(* IEC 61131-3 sources: AXOpen/src/components.dukane.welders/ctrl/src/Axo_IQ_SeriesWelder (part 2) *)

        METHOD PRIVATE ByteArray_TO_buf4
            VAR_INPUT
                array_buffer : ARRAY[0..253] OF BYTE;
            END_VAR
            VAR_IN_OUT
                buf4 : Axo_IQ_SeriesWelder_data4_200bytes;
            END_VAR
			buf4.Weld2Distance.Enable._0 						    :=   array_buffer[  0].%X0;
			buf4.Weld2Distance.Enable._1 						    :=   array_buffer[  0].%X1;
			buf4.Weld2Distance.Enable._2 						    :=   array_buffer[  0].%X2;
			buf4.Weld2Distance.Enable._3 						    :=   array_buffer[  0].%X3;
			buf4.Weld2Distance.Enable._4 						    :=   array_buffer[  0].%X4;
			buf4.Weld2Distance.Enable._5 						    :=   array_buffer[  0].%X5;
			buf4.Weld2Distance.Enable._6 						    :=   array_buffer[  0].%X6;
			buf4.Weld2Distance.Enable._7 						    :=   array_buffer[  0].%X7;
			buf4.Weld2Distance.Enable._8 						    :=   array_buffer[  1].%X0;
			buf4.Weld2Distance.Enable._9 						    :=   array_buffer[  1].%X1;
			buf4.Weld2Distance.Enable._10 					        :=   array_buffer[  1].%X2;
			buf4.Weld2Distance.Enable._11 					        :=   array_buffer[  1].%X3;
			buf4.Weld2Distance.Enable._12 					        :=   array_buffer[  1].%X4;
			buf4.Weld2Distance.Enable._13 					        :=   array_buffer[  1].%X5;
			buf4.Weld2Distance.Enable._14 					        :=   array_buffer[  1].%X6;
			buf4.Weld2Distance.Enable._15 					        :=   array_buffer[  1].%X7;
			buf4.Weld2Distance.Enable._16 					        :=   array_buffer[  2].%X0;
			buf4.Weld2Distance.Enable._17 					        :=   array_buffer[  2].%X1;
			buf4.Weld2Distance.Enable._18 					        :=   array_buffer[  2].%X2;
			buf4.Weld2Distance.Enable._19 					        :=   array_buffer[  2].%X3;
			buf4.Weld2Distance.Enable._20 					        :=   array_buffer[  2].%X4;
			buf4.Weld2Distance.Enable._21 					        :=   array_buffer[  2].%X5;
			buf4.Weld2Distance.Enable._22 					        :=   array_buffer[  2].%X6;
			buf4.Weld2Distance.Enable._23 					        :=   array_buffer[  2].%X7;
			buf4.Weld2Distance.Enable.LowerBad_1 				    :=   array_buffer[  3].%X0;
			buf4.Weld2Distance.Enable.LowerSuspect_1 			    :=   array_buffer[  3].%X1;
			buf4.Weld2Distance.Enable.UpperSuspect_1			    :=   array_buffer[  3].%X2;
			buf4.Weld2Distance.Enable.UpperBad_1 				    :=   array_buffer[  3].%X3;
			buf4.Weld2Distance.Enable.Display_1 				    :=   array_buffer[  3].%X4;
			buf4.Weld2Distance.Enable._29 					        :=   array_buffer[  3].%X5;
			buf4.Weld2Distance.Enable._30 					        :=   array_buffer[  3].%X6;
			buf4.Weld2Distance.Enable._31 					        :=   array_buffer[  3].%X7;
			buf4.Weld2Distance.LowerBad:=           TO_DINT(SHL(TO_DWORD(array_buffer[  4]), UINT#24) OR
															SHL(TO_DWORD(array_buffer[  5]), UINT#16) OR
															SHL(TO_DWORD(array_buffer[  6]),  UINT#8) OR
																TO_DWORD(array_buffer[  7]));
			buf4.Weld2Distance.LowerSuspect:=       TO_DINT(SHL(TO_DWORD(array_buffer[  8]), UINT#24) OR
															SHL(TO_DWORD(array_buffer[  9]), UINT#16) OR
															SHL(TO_DWORD(array_buffer[ 10]),  UINT#8) OR
																TO_DWORD(array_buffer[ 11]));
			buf4.Weld2Distance.UpperSuspect:=       TO_DINT(SHL(TO_DWORD(array_buffer[ 12]), UINT#24) OR
															SHL(TO_DWORD(array_buffer[ 13]), UINT#16) OR
															SHL(TO_DWORD(array_buffer[ 14]),  UINT#8) OR
																TO_DWORD(array_buffer[ 15]));
			buf4.Weld2Distance.UpperBad:=           TO_DINT(SHL(TO_DWORD(array_buffer[ 16]), UINT#24) OR
															SHL(TO_DWORD(array_buffer[ 17]), UINT#16) OR
															SHL(TO_DWORD(array_buffer[ 18]),  UINT#8) OR
																TO_DWORD(array_buffer[ 19]));
			buf4.Weld2Position.Enable._0 					        :=   array_buffer[ 20].%X0;
			buf4.Weld2Position.Enable._1 					        :=   array_buffer[ 20].%X1;
			buf4.Weld2Position.Enable._2 					        :=   array_buffer[ 20].%X2;
			buf4.Weld2Position.Enable._3 					        :=   array_buffer[ 20].%X3;
			buf4.Weld2Position.Enable._4 					        :=   array_buffer[ 20].%X4;
			buf4.Weld2Position.Enable._5 					        :=   array_buffer[ 20].%X5;
			buf4.Weld2Position.Enable._6 					        :=   array_buffer[ 20].%X6;
			buf4.Weld2Position.Enable._7 					        :=   array_buffer[ 20].%X7;
			buf4.Weld2Position.Enable._8 					        :=   array_buffer[ 21].%X0;
			buf4.Weld2Position.Enable._9 					        :=   array_buffer[ 21].%X1;
			buf4.Weld2Position.Enable._10 				            :=   array_buffer[ 21].%X2;
			buf4.Weld2Position.Enable._11 				            :=   array_buffer[ 21].%X3;
			buf4.Weld2Position.Enable._12 				            :=   array_buffer[ 21].%X4;
			buf4.Weld2Position.Enable._13 				            :=   array_buffer[ 21].%X5;
			buf4.Weld2Position.Enable._14 				            :=   array_buffer[ 21].%X6;
			buf4.Weld2Position.Enable._15 				            :=   array_buffer[ 21].%X7;
			buf4.Weld2Position.Enable._16 				            :=   array_buffer[ 22].%X0;
			buf4.Weld2Position.Enable._17 				            :=   array_buffer[ 22].%X1;
			buf4.Weld2Position.Enable._18 				            :=   array_buffer[ 22].%X2;
			buf4.Weld2Position.Enable._19 				            :=   array_buffer[ 22].%X3;
			buf4.Weld2Position.Enable._20 				            :=   array_buffer[ 22].%X4;
			buf4.Weld2Position.Enable._21 				            :=   array_buffer[ 22].%X5;
			buf4.Weld2Position.Enable._22 				            :=   array_buffer[ 22].%X6;
			buf4.Weld2Position.Enable._23 				            :=   array_buffer[ 22].%X7;
			buf4.Weld2Position.Enable.LowerBad_1 			        :=   array_buffer[ 23].%X0;
			buf4.Weld2Position.Enable.LowerSuspect_1 		        :=   array_buffer[ 23].%X1;
			buf4.Weld2Position.Enable.UpperSuspect_1		        :=   array_buffer[ 23].%X2;
			buf4.Weld2Position.Enable.UpperBad_1 				    :=   array_buffer[ 23].%X3;
			buf4.Weld2Position.Enable.Display_1 				    :=   array_buffer[ 23].%X4;
			buf4.Weld2Position.Enable._29 					        :=   array_buffer[ 23].%X5;
			buf4.Weld2Position.Enable._30 					        :=   array_buffer[ 23].%X6;
			buf4.Weld2Position.Enable._31 					        :=   array_buffer[ 23].%X7;
			buf4.Weld2Position.LowerBad:=           TO_DINT(SHL(TO_DWORD(array_buffer[ 24]), UINT#24) OR
															SHL(TO_DWORD(array_buffer[ 25]), UINT#16) OR
															SHL(TO_DWORD(array_buffer[ 26]),  UINT#8) OR
																TO_DWORD(array_buffer[ 27]));
			buf4.Weld2Position.LowerSuspect:=       TO_DINT(SHL(TO_DWORD(array_buffer[ 28]), UINT#24) OR
															SHL(TO_DWORD(array_buffer[ 29]), UINT#16) OR
															SHL(TO_DWORD(array_buffer[ 30]),  UINT#8) OR
																TO_DWORD(array_buffer[ 31]));
			buf4.Weld2Position.UpperSuspect:=       TO_DINT(SHL(TO_DWORD(array_buffer[ 32]), UINT#24) OR
															SHL(TO_DWORD(array_buffer[ 33]), UINT#16) OR
															SHL(TO_DWORD(array_buffer[ 34]),  UINT#8) OR
																TO_DWORD(array_buffer[ 35]));
			buf4.Weld2Position.UpperBad:=           TO_DINT(SHL(TO_DWORD(array_buffer[ 36]), UINT#24) OR
															SHL(TO_DWORD(array_buffer[ 37]), UINT#16) OR
															SHL(TO_DWORD(array_buffer[ 38]),  UINT#8) OR
																TO_DWORD(array_buffer[ 39]));
			buf4.TotalWeldTime.Enable._0 					        :=   array_buffer[ 40].%X0;
			buf4.TotalWeldTime.Enable._1 					        :=   array_buffer[ 40].%X1;
			buf4.TotalWeldTime.Enable._2 					        :=   array_buffer[ 40].%X2;
			buf4.TotalWeldTime.Enable._3 					        :=   array_buffer[ 40].%X3;
			buf4.TotalWeldTime.Enable._4 					        :=   array_buffer[ 40].%X4;
			buf4.TotalWeldTime.Enable._5 					        :=   array_buffer[ 40].%X5;
			buf4.TotalWeldTime.Enable._6 					        :=   array_buffer[ 40].%X6;
			buf4.TotalWeldTime.Enable._7 					        :=   array_buffer[ 40].%X7;
			buf4.TotalWeldTime.Enable._8 					        :=   array_buffer[ 41].%X0;
			buf4.TotalWeldTime.Enable._9 					        :=   array_buffer[ 41].%X1;
			buf4.TotalWeldTime.Enable._10 				            :=   array_buffer[ 41].%X2;
			buf4.TotalWeldTime.Enable._11 				            :=   array_buffer[ 41].%X3;
			buf4.TotalWeldTime.Enable._12 				            :=   array_buffer[ 41].%X4;
			buf4.TotalWeldTime.Enable._13 				            :=   array_buffer[ 41].%X5;
			buf4.TotalWeldTime.Enable._14 				            :=   array_buffer[ 41].%X6;
			buf4.TotalWeldTime.Enable._15 				            :=   array_buffer[ 41].%X7;
			buf4.TotalWeldTime.Enable._16 				            :=   array_buffer[ 42].%X0;
			buf4.TotalWeldTime.Enable._17 				            :=   array_buffer[ 42].%X1;
			buf4.TotalWeldTime.Enable._18 				            :=   array_buffer[ 42].%X2;
			buf4.TotalWeldTime.Enable._19 				            :=   array_buffer[ 42].%X3;
			buf4.TotalWeldTime.Enable._20 				            :=   array_buffer[ 42].%X4;
			buf4.TotalWeldTime.Enable._21 				            :=   array_buffer[ 42].%X5;
			buf4.TotalWeldTime.Enable._22 				            :=   array_buffer[ 42].%X6;
			buf4.TotalWeldTime.Enable._23 				            :=   array_buffer[ 42].%X7;
			buf4.TotalWeldTime.Enable.LowerBad_1 			        :=   array_buffer[ 43].%X0;
			buf4.TotalWeldTime.Enable.LowerSuspect_1 		        :=   array_buffer[ 43].%X1;
			buf4.TotalWeldTime.Enable.UpperSuspect_1		        :=   array_buffer[ 43].%X2;
			buf4.TotalWeldTime.Enable.UpperBad_1 			        :=   array_buffer[ 43].%X3;
			buf4.TotalWeldTime.Enable.Display_1 				    :=   array_buffer[ 43].%X4;
			buf4.TotalWeldTime.Enable._29 					        :=   array_buffer[ 43].%X5;
			buf4.TotalWeldTime.Enable._30 					        :=   array_buffer[ 43].%X6;
			buf4.TotalWeldTime.Enable._31 					        :=   array_buffer[ 43].%X7;
			buf4.TotalWeldTime.LowerBad:=           TO_DINT(SHL(TO_DWORD(array_buffer[ 44]), UINT#24) OR
															SHL(TO_DWORD(array_buffer[ 45]), UINT#16) OR
															SHL(TO_DWORD(array_buffer[ 46]),  UINT#8) OR
																TO_DWORD(array_buffer[ 47]));
			buf4.TotalWeldTime.LowerSuspect:=       TO_DINT(SHL(TO_DWORD(array_buffer[ 48]), UINT#24) OR
															SHL(TO_DWORD(array_buffer[ 49]), UINT#16) OR
															SHL(TO_DWORD(array_buffer[ 50]),  UINT#8) OR
																TO_DWORD(array_buffer[ 51]));
			buf4.TotalWeldTime.UpperSuspect:=       TO_DINT(SHL(TO_DWORD(array_buffer[ 52]), UINT#24) OR
															SHL(TO_DWORD(array_buffer[ 53]), UINT#16) OR
															SHL(TO_DWORD(array_buffer[ 54]),  UINT#8) OR
																TO_DWORD(array_buffer[ 55]));
			buf4.TotalWeldTime.UpperBad:=           TO_DINT(SHL(TO_DWORD(array_buffer[ 56]), UINT#24) OR
															SHL(TO_DWORD(array_buffer[ 57]), UINT#16) OR
															SHL(TO_DWORD(array_buffer[ 58]),  UINT#8) OR
																TO_DWORD(array_buffer[ 59]));
			buf4.TotalWeldEnergy.Enable._0 				            :=   array_buffer[ 60].%X0;
			buf4.TotalWeldEnergy.Enable._1 				            :=   array_buffer[ 60].%X1;
			buf4.TotalWeldEnergy.Enable._2 				            :=   array_buffer[ 60].%X2;
			buf4.TotalWeldEnergy.Enable._3 				            :=   array_buffer[ 60].%X3;
			buf4.TotalWeldEnergy.Enable._4 				            :=   array_buffer[ 60].%X4;
			buf4.TotalWeldEnergy.Enable._5 				            :=   array_buffer[ 60].%X5;
			buf4.TotalWeldEnergy.Enable._6 				            :=   array_buffer[ 60].%X6;
			buf4.TotalWeldEnergy.Enable._7 				            :=   array_buffer[ 60].%X7;
			buf4.TotalWeldEnergy.Enable._8 				            :=   array_buffer[ 61].%X0;
			buf4.TotalWeldEnergy.Enable._9 				            :=   array_buffer[ 61].%X1;
			buf4.TotalWeldEnergy.Enable._10 				        :=   array_buffer[ 61].%X2;
			buf4.TotalWeldEnergy.Enable._11 				        :=   array_buffer[ 61].%X3;
			buf4.TotalWeldEnergy.Enable._12 				        :=   array_buffer[ 61].%X4;
			buf4.TotalWeldEnergy.Enable._13 				        :=   array_buffer[ 61].%X5;
			buf4.TotalWeldEnergy.Enable._14 				        :=   array_buffer[ 61].%X6;
			buf4.TotalWeldEnergy.Enable._15 				        :=   array_buffer[ 61].%X7;
			buf4.TotalWeldEnergy.Enable._16 				        :=   array_buffer[ 62].%X0;
			buf4.TotalWeldEnergy.Enable._17 				        :=   array_buffer[ 62].%X1;
			buf4.TotalWeldEnergy.Enable._18 				        :=   array_buffer[ 62].%X2;
			buf4.TotalWeldEnergy.Enable._19 				        :=   array_buffer[ 62].%X3;
			buf4.TotalWeldEnergy.Enable._20 				        :=   array_buffer[ 62].%X4;
			buf4.TotalWeldEnergy.Enable._21 				        :=   array_buffer[ 62].%X5;
			buf4.TotalWeldEnergy.Enable._22 				        :=   array_buffer[ 62].%X6;
			buf4.TotalWeldEnergy.Enable._23 				        :=   array_buffer[ 62].%X7;
			buf4.TotalWeldEnergy.Enable.LowerBad_1 		            :=   array_buffer[ 63].%X0;
			buf4.TotalWeldEnergy.Enable.LowerSuspect_1 	            :=   array_buffer[ 63].%X1;
			buf4.TotalWeldEnergy.Enable.UpperSuspect_1		        :=   array_buffer[ 63].%X2;
			buf4.TotalWeldEnergy.Enable.UpperBad_1 		            :=   array_buffer[ 63].%X3;
			buf4.TotalWeldEnergy.Enable.Display_1 			        :=   array_buffer[ 63].%X4;
			buf4.TotalWeldEnergy.Enable._29 				        :=   array_buffer[ 63].%X5;
			buf4.TotalWeldEnergy.Enable._30 				        :=   array_buffer[ 63].%X6;
			buf4.TotalWeldEnergy.Enable._31 				        :=   array_buffer[ 63].%X7;
			buf4.TotalWeldEnergy.LowerBad:=         TO_DINT(SHL(TO_DWORD(array_buffer[ 64]), UINT#24) OR
															SHL(TO_DWORD(array_buffer[ 65]), UINT#16) OR
															SHL(TO_DWORD(array_buffer[ 66]),  UINT#8) OR
																TO_DWORD(array_buffer[ 67]));
			buf4.TotalWeldEnergy.LowerSuspect:=     TO_DINT(SHL(TO_DWORD(array_buffer[ 68]), UINT#24) OR
															SHL(TO_DWORD(array_buffer[ 69]), UINT#16) OR
															SHL(TO_DWORD(array_buffer[ 70]),  UINT#8) OR
																TO_DWORD(array_buffer[ 71]));
			buf4.TotalWeldEnergy.UpperSuspect:=     TO_DINT(SHL(TO_DWORD(array_buffer[ 72]), UINT#24) OR
															SHL(TO_DWORD(array_buffer[ 73]), UINT#16) OR
															SHL(TO_DWORD(array_buffer[ 74]),  UINT#8) OR
																TO_DWORD(array_buffer[ 75]));
			buf4.TotalWeldEnergy.UpperBad:=         TO_DINT(SHL(TO_DWORD(array_buffer[ 76]), UINT#24) OR
															SHL(TO_DWORD(array_buffer[ 77]), UINT#16) OR
															SHL(TO_DWORD(array_buffer[ 78]),  UINT#8) OR
																TO_DWORD(array_buffer[ 79]));
			buf4.TotalWeldDistance.Enable._0 				        :=   array_buffer[ 80].%X0;
			buf4.TotalWeldDistance.Enable._1 				        :=   array_buffer[ 80].%X1;
			buf4.TotalWeldDistance.Enable._2 				        :=   array_buffer[ 80].%X2;
			buf4.TotalWeldDistance.Enable._3 				        :=   array_buffer[ 80].%X3;
			buf4.TotalWeldDistance.Enable._4 				        :=   array_buffer[ 80].%X4;
			buf4.TotalWeldDistance.Enable._5 				        :=   array_buffer[ 80].%X5;
			buf4.TotalWeldDistance.Enable._6 				        :=   array_buffer[ 80].%X6;
			buf4.TotalWeldDistance.Enable._7 				        :=   array_buffer[ 80].%X7;
			buf4.TotalWeldDistance.Enable._8 				        :=   array_buffer[ 81].%X0;
			buf4.TotalWeldDistance.Enable._9 				        :=   array_buffer[ 81].%X1;
			buf4.TotalWeldDistance.Enable._10 				        :=   array_buffer[ 81].%X2;
			buf4.TotalWeldDistance.Enable._11 				        :=   array_buffer[ 81].%X3;
			buf4.TotalWeldDistance.Enable._12 				        :=   array_buffer[ 81].%X4;
			buf4.TotalWeldDistance.Enable._13 				        :=   array_buffer[ 81].%X5;
			buf4.TotalWeldDistance.Enable._14 				        :=   array_buffer[ 81].%X6;
			buf4.TotalWeldDistance.Enable._15 				        :=   array_buffer[ 81].%X7;
			buf4.TotalWeldDistance.Enable._16 				        :=   array_buffer[ 82].%X0;
			buf4.TotalWeldDistance.Enable._17 				        :=   array_buffer[ 82].%X1;
			buf4.TotalWeldDistance.Enable._18 				        :=   array_buffer[ 82].%X2;
			buf4.TotalWeldDistance.Enable._19 				        :=   array_buffer[ 82].%X3;
			buf4.TotalWeldDistance.Enable._20 				        :=   array_buffer[ 82].%X4;
			buf4.TotalWeldDistance.Enable._21 				        :=   array_buffer[ 82].%X5;
			buf4.TotalWeldDistance.Enable._22 				        :=   array_buffer[ 82].%X6;
			buf4.TotalWeldDistance.Enable._23 				        :=   array_buffer[ 82].%X7;
			buf4.TotalWeldDistance.Enable.LowerBad_1 		        :=   array_buffer[ 83].%X0;
			buf4.TotalWeldDistance.Enable.LowerSuspect_1 	        :=   array_buffer[ 83].%X1;
			buf4.TotalWeldDistance.Enable.UpperSuspect_1		    :=   array_buffer[ 83].%X2;
			buf4.TotalWeldDistance.Enable.UpperBad_1 		        :=   array_buffer[ 83].%X3;
			buf4.TotalWeldDistance.Enable.Display_1 			    :=   array_buffer[ 83].%X4;
			buf4.TotalWeldDistance.Enable._29 				        :=   array_buffer[ 83].%X5;
			buf4.TotalWeldDistance.Enable._30 				        :=   array_buffer[ 83].%X6;
			buf4.TotalWeldDistance.Enable._31 				        :=   array_buffer[ 83].%X7;
			buf4.TotalWeldDistance.LowerBad:=       TO_DINT(SHL(TO_DWORD(array_buffer[ 84]), UINT#24) OR
															SHL(TO_DWORD(array_buffer[ 85]), UINT#16) OR
															SHL(TO_DWORD(array_buffer[ 86]),  UINT#8) OR
																TO_DWORD(array_buffer[ 87]));
			buf4.TotalWeldDistance.LowerSuspect:=   TO_DINT(SHL(TO_DWORD(array_buffer[ 88]), UINT#24) OR
															SHL(TO_DWORD(array_buffer[ 89]), UINT#16) OR
															SHL(TO_DWORD(array_buffer[ 90]),  UINT#8) OR
																TO_DWORD(array_buffer[ 91]));
			buf4.TotalWeldDistance.UpperSuspect:=   TO_DINT(SHL(TO_DWORD(array_buffer[ 92]), UINT#24) OR
															SHL(TO_DWORD(array_buffer[ 93]), UINT#16) OR
															SHL(TO_DWORD(array_buffer[ 94]),  UINT#8) OR
																TO_DWORD(array_buffer[ 95]));
			buf4.TotalWeldDistance.UpperBad:=       TO_DINT(SHL(TO_DWORD(array_buffer[ 96]), UINT#24) OR
															SHL(TO_DWORD(array_buffer[ 97]), UINT#16) OR
															SHL(TO_DWORD(array_buffer[ 98]),  UINT#8) OR
																TO_DWORD(array_buffer[ 99]));
			buf4.DynamicHoldTime.Enable._0 				            :=   array_buffer[100].%X0;
			buf4.DynamicHoldTime.Enable._1 				            :=   array_buffer[100].%X1;
			buf4.DynamicHoldTime.Enable._2 				            :=   array_buffer[100].%X2;
			buf4.DynamicHoldTime.Enable._3 				            :=   array_buffer[100].%X3;
			buf4.DynamicHoldTime.Enable._4 				            :=   array_buffer[100].%X4;
			buf4.DynamicHoldTime.Enable._5 				            :=   array_buffer[100].%X5;
			buf4.DynamicHoldTime.Enable._6 				            :=   array_buffer[100].%X6;
			buf4.DynamicHoldTime.Enable._7 				            :=   array_buffer[100].%X7;
			buf4.DynamicHoldTime.Enable._8 				            :=   array_buffer[101].%X0;
			buf4.DynamicHoldTime.Enable._9 				            :=   array_buffer[101].%X1;
			buf4.DynamicHoldTime.Enable._10 				        :=   array_buffer[101].%X2;
			buf4.DynamicHoldTime.Enable._11 				        :=   array_buffer[101].%X3;
			buf4.DynamicHoldTime.Enable._12 				        :=   array_buffer[101].%X4;
			buf4.DynamicHoldTime.Enable._13 				        :=   array_buffer[101].%X5;
			buf4.DynamicHoldTime.Enable._14 				        :=   array_buffer[101].%X6;
			buf4.DynamicHoldTime.Enable._15 				        :=   array_buffer[101].%X7;
			buf4.DynamicHoldTime.Enable._16 				        :=   array_buffer[102].%X0;
			buf4.DynamicHoldTime.Enable._17 				        :=   array_buffer[102].%X1;
			buf4.DynamicHoldTime.Enable._18 				        :=   array_buffer[102].%X2;
			buf4.DynamicHoldTime.Enable._19 				        :=   array_buffer[102].%X3;
			buf4.DynamicHoldTime.Enable._20 				        :=   array_buffer[102].%X4;
			buf4.DynamicHoldTime.Enable._21 				        :=   array_buffer[102].%X5;
			buf4.DynamicHoldTime.Enable._22 				        :=   array_buffer[102].%X6;
			buf4.DynamicHoldTime.Enable._23 				        :=   array_buffer[102].%X7;
			buf4.DynamicHoldTime.Enable.LowerBad_1 		            :=   array_buffer[103].%X0;
			buf4.DynamicHoldTime.Enable.LowerSuspect_1 	            :=   array_buffer[103].%X1;
			buf4.DynamicHoldTime.Enable.UpperSuspect_1		        :=   array_buffer[103].%X2;
			buf4.DynamicHoldTime.Enable.UpperBad_1 		            :=   array_buffer[103].%X3;
			buf4.DynamicHoldTime.Enable.Display_1 			        :=   array_buffer[103].%X4;
			buf4.DynamicHoldTime.Enable._29 				        :=   array_buffer[103].%X5;
			buf4.DynamicHoldTime.Enable._30 				        :=   array_buffer[103].%X6;
			buf4.DynamicHoldTime.Enable._31 				        :=   array_buffer[103].%X7;
			buf4.DynamicHoldTime.LowerBad:=         TO_DINT(SHL(TO_DWORD(array_buffer[104]), UINT#24) OR
															SHL(TO_DWORD(array_buffer[105]), UINT#16) OR
															SHL(TO_DWORD(array_buffer[106]),  UINT#8) OR
																TO_DWORD(array_buffer[107]));
			buf4.DynamicHoldTime.LowerSuspect:=     TO_DINT(SHL(TO_DWORD(array_buffer[108]), UINT#24) OR
															SHL(TO_DWORD(array_buffer[109]), UINT#16) OR
															SHL(TO_DWORD(array_buffer[110]),  UINT#8) OR
																TO_DWORD(array_buffer[111]));
			buf4.DynamicHoldTime.UpperSuspect:=     TO_DINT(SHL(TO_DWORD(array_buffer[112]), UINT#24) OR
															SHL(TO_DWORD(array_buffer[113]), UINT#16) OR
															SHL(TO_DWORD(array_buffer[114]),  UINT#8) OR
																TO_DWORD(array_buffer[115]));
			buf4.DynamicHoldTime.UpperBad:=         TO_DINT(SHL(TO_DWORD(array_buffer[116]), UINT#24) OR
															SHL(TO_DWORD(array_buffer[117]), UINT#16) OR
															SHL(TO_DWORD(array_buffer[118]),  UINT#8) OR
																TO_DWORD(array_buffer[119]));
			buf4.DynamicHoldDistance.Enable._0 				        :=   array_buffer[120].%X0;
			buf4.DynamicHoldDistance.Enable._1 				        :=   array_buffer[120].%X1;
			buf4.DynamicHoldDistance.Enable._2 				        :=   array_buffer[120].%X2;
			buf4.DynamicHoldDistance.Enable._3 				        :=   array_buffer[120].%X3;
			buf4.DynamicHoldDistance.Enable._4 				        :=   array_buffer[120].%X4;
			buf4.DynamicHoldDistance.Enable._5 				        :=   array_buffer[120].%X5;
			buf4.DynamicHoldDistance.Enable._6 				        :=   array_buffer[120].%X6;
			buf4.DynamicHoldDistance.Enable._7 				        :=   array_buffer[120].%X7;
			buf4.DynamicHoldDistance.Enable._8 				        :=   array_buffer[121].%X0;
			buf4.DynamicHoldDistance.Enable._9 				        :=   array_buffer[121].%X1;
			buf4.DynamicHoldDistance.Enable._10 				    :=   array_buffer[121].%X2;
			buf4.DynamicHoldDistance.Enable._11 				    :=   array_buffer[121].%X3;
			buf4.DynamicHoldDistance.Enable._12 				    :=   array_buffer[121].%X4;
			buf4.DynamicHoldDistance.Enable._13 				    :=   array_buffer[121].%X5;
			buf4.DynamicHoldDistance.Enable._14 				    :=   array_buffer[121].%X6;
			buf4.DynamicHoldDistance.Enable._15 				    :=   array_buffer[121].%X7;
			buf4.DynamicHoldDistance.Enable._16 				    :=   array_buffer[122].%X0;
			buf4.DynamicHoldDistance.Enable._17 				    :=   array_buffer[122].%X1;
			buf4.DynamicHoldDistance.Enable._18 				    :=   array_buffer[122].%X2;
			buf4.DynamicHoldDistance.Enable._19 				    :=   array_buffer[122].%X3;
			buf4.DynamicHoldDistance.Enable._20 				    :=   array_buffer[122].%X4;
			buf4.DynamicHoldDistance.Enable._21 				    :=   array_buffer[122].%X5;
			buf4.DynamicHoldDistance.Enable._22 				    :=   array_buffer[122].%X6;
			buf4.DynamicHoldDistance.Enable._23 				    :=   array_buffer[122].%X7;
			buf4.DynamicHoldDistance.Enable.LowerBad_1 		        :=   array_buffer[123].%X0;
			buf4.DynamicHoldDistance.Enable.LowerSuspect_1 	        :=   array_buffer[123].%X1;
			buf4.DynamicHoldDistance.Enable.UpperSuspect_1		    :=   array_buffer[123].%X2;
			buf4.DynamicHoldDistance.Enable.UpperBad_1 		        :=   array_buffer[123].%X3;
			buf4.DynamicHoldDistance.Enable.Display_1 			    :=   array_buffer[123].%X4;
			buf4.DynamicHoldDistance.Enable._29 				    :=   array_buffer[123].%X5;
			buf4.DynamicHoldDistance.Enable._30 				    :=   array_buffer[123].%X6;
			buf4.DynamicHoldDistance.Enable._31 				    :=   array_buffer[123].%X7;
			buf4.DynamicHoldDistance.LowerBad:=     TO_DINT(SHL(TO_DWORD(array_buffer[124]), UINT#24) OR
															SHL(TO_DWORD(array_buffer[125]), UINT#16) OR
															SHL(TO_DWORD(array_buffer[126]),  UINT#8) OR
																TO_DWORD(array_buffer[127]));
			buf4.DynamicHoldDistance.LowerSuspect:= TO_DINT(SHL(TO_DWORD(array_buffer[128]), UINT#24) OR
															SHL(TO_DWORD(array_buffer[129]), UINT#16) OR
															SHL(TO_DWORD(array_buffer[130]),  UINT#8) OR
																TO_DWORD(array_buffer[131]));
			buf4.DynamicHoldDistance.UpperSuspect:= TO_DINT(SHL(TO_DWORD(array_buffer[132]), UINT#24) OR
															SHL(TO_DWORD(array_buffer[133]), UINT#16) OR
															SHL(TO_DWORD(array_buffer[134]),  UINT#8) OR
																TO_DWORD(array_buffer[135]));
			buf4.DynamicHoldDistance.UpperBad:=     TO_DINT(SHL(TO_DWORD(array_buffer[136]), UINT#24) OR
															SHL(TO_DWORD(array_buffer[137]), UINT#16) OR
															SHL(TO_DWORD(array_buffer[138]),  UINT#8) OR
																TO_DWORD(array_buffer[139]));
			buf4.TotalCycleTime.Enable._0 				            :=   array_buffer[140].%X0;
			buf4.TotalCycleTime.Enable._1 				            :=   array_buffer[140].%X1;
			buf4.TotalCycleTime.Enable._2 				            :=   array_buffer[140].%X2;
			buf4.TotalCycleTime.Enable._3 				            :=   array_buffer[140].%X3;
			buf4.TotalCycleTime.Enable._4 				            :=   array_buffer[140].%X4;
			buf4.TotalCycleTime.Enable._5 				            :=   array_buffer[140].%X5;
			buf4.TotalCycleTime.Enable._6 				            :=   array_buffer[140].%X6;
			buf4.TotalCycleTime.Enable._7 				            :=   array_buffer[140].%X7;
			buf4.TotalCycleTime.Enable._8 				            :=   array_buffer[141].%X0;
			buf4.TotalCycleTime.Enable._9 				            :=   array_buffer[141].%X1;
			buf4.TotalCycleTime.Enable._10 				            :=   array_buffer[141].%X2;
			buf4.TotalCycleTime.Enable._11 				            :=   array_buffer[141].%X3;
			buf4.TotalCycleTime.Enable._12 				            :=   array_buffer[141].%X4;
			buf4.TotalCycleTime.Enable._13 				            :=   array_buffer[141].%X5;
			buf4.TotalCycleTime.Enable._14 				            :=   array_buffer[141].%X6;
			buf4.TotalCycleTime.Enable._15 				            :=   array_buffer[141].%X7;
			buf4.TotalCycleTime.Enable._16 				            :=   array_buffer[142].%X0;
			buf4.TotalCycleTime.Enable._17 				            :=   array_buffer[142].%X1;
			buf4.TotalCycleTime.Enable._18 				            :=   array_buffer[142].%X2;
			buf4.TotalCycleTime.Enable._19 				            :=   array_buffer[142].%X3;
			buf4.TotalCycleTime.Enable._20 				            :=   array_buffer[142].%X4;
			buf4.TotalCycleTime.Enable._21 				            :=   array_buffer[142].%X5;
			buf4.TotalCycleTime.Enable._22 				            :=   array_buffer[142].%X6;
			buf4.TotalCycleTime.Enable._23 				            :=   array_buffer[142].%X7;
			buf4.TotalCycleTime.Enable.LowerBad_1 		            :=   array_buffer[143].%X0;
			buf4.TotalCycleTime.Enable.LowerSuspect_1 	            :=   array_buffer[143].%X1;
			buf4.TotalCycleTime.Enable.UpperSuspect_1		        :=   array_buffer[143].%X2;
			buf4.TotalCycleTime.Enable.UpperBad_1 		            :=   array_buffer[143].%X3;
			buf4.TotalCycleTime.Enable.Display_1 			        :=   array_buffer[143].%X4;
			buf4.TotalCycleTime.Enable._29 				            :=   array_buffer[143].%X5;
			buf4.TotalCycleTime.Enable._30 				            :=   array_buffer[143].%X6;
			buf4.TotalCycleTime.Enable._31 				            :=   array_buffer[143].%X7;
			buf4.TotalCycleTime.LowerBad:=          TO_DINT(SHL(TO_DWORD(array_buffer[144]), UINT#24) OR
															SHL(TO_DWORD(array_buffer[145]), UINT#16) OR
															SHL(TO_DWORD(array_buffer[146]),  UINT#8) OR
																TO_DWORD(array_buffer[147]));
			buf4.TotalCycleTime.LowerSuspect:=      TO_DINT(SHL(TO_DWORD(array_buffer[148]), UINT#24) OR
															SHL(TO_DWORD(array_buffer[149]), UINT#16) OR
															SHL(TO_DWORD(array_buffer[150]),  UINT#8) OR
																TO_DWORD(array_buffer[151]));
			buf4.TotalCycleTime.UpperSuspect:=      TO_DINT(SHL(TO_DWORD(array_buffer[152]), UINT#24) OR
															SHL(TO_DWORD(array_buffer[153]), UINT#16) OR
															SHL(TO_DWORD(array_buffer[154]),  UINT#8) OR
																TO_DWORD(array_buffer[155]));
			buf4.TotalCycleTime.UpperBad:=          TO_DINT(SHL(TO_DWORD(array_buffer[156]), UINT#24) OR
															SHL(TO_DWORD(array_buffer[157]), UINT#16) OR
															SHL(TO_DWORD(array_buffer[158]),  UINT#8) OR
																TO_DWORD(array_buffer[159]));
			buf4.FinalHoldPosition.Enable._0 				        :=   array_buffer[160].%X0;
			buf4.FinalHoldPosition.Enable._1 				        :=   array_buffer[160].%X1;
			buf4.FinalHoldPosition.Enable._2 				        :=   array_buffer[160].%X2;
			buf4.FinalHoldPosition.Enable._3 				        :=   array_buffer[160].%X3;
			buf4.FinalHoldPosition.Enable._4 				        :=   array_buffer[160].%X4;
			buf4.FinalHoldPosition.Enable._5 				        :=   array_buffer[160].%X5;
			buf4.FinalHoldPosition.Enable._6 				        :=   array_buffer[160].%X6;
			buf4.FinalHoldPosition.Enable._7 				        :=   array_buffer[160].%X7;
			buf4.FinalHoldPosition.Enable._8 				        :=   array_buffer[161].%X0;
			buf4.FinalHoldPosition.Enable._9 				        :=   array_buffer[161].%X1;
			buf4.FinalHoldPosition.Enable._10 				        :=   array_buffer[161].%X2;
			buf4.FinalHoldPosition.Enable._11 				        :=   array_buffer[161].%X3;
			buf4.FinalHoldPosition.Enable._12 				        :=   array_buffer[161].%X4;
			buf4.FinalHoldPosition.Enable._13 				        :=   array_buffer[161].%X5;
			buf4.FinalHoldPosition.Enable._14 				        :=   array_buffer[161].%X6;
			buf4.FinalHoldPosition.Enable._15 				        :=   array_buffer[161].%X7;
			buf4.FinalHoldPosition.Enable._16 				        :=   array_buffer[162].%X0;
			buf4.FinalHoldPosition.Enable._17 				        :=   array_buffer[162].%X1;
			buf4.FinalHoldPosition.Enable._18 				        :=   array_buffer[162].%X2;
			buf4.FinalHoldPosition.Enable._19 				        :=   array_buffer[162].%X3;
			buf4.FinalHoldPosition.Enable._20 				        :=   array_buffer[162].%X4;
			buf4.FinalHoldPosition.Enable._21 				        :=   array_buffer[162].%X5;
			buf4.FinalHoldPosition.Enable._22 				        :=   array_buffer[162].%X6;
			buf4.FinalHoldPosition.Enable._23 				        :=   array_buffer[162].%X7;
			buf4.FinalHoldPosition.Enable.LowerBad_1 		        :=   array_buffer[163].%X0;
			buf4.FinalHoldPosition.Enable.LowerSuspect_1 	        :=   array_buffer[163].%X1;
			buf4.FinalHoldPosition.Enable.UpperSuspect_1		    :=   array_buffer[163].%X2;
			buf4.FinalHoldPosition.Enable.UpperBad_1 		        :=   array_buffer[163].%X3;
			buf4.FinalHoldPosition.Enable.Display_1 			    :=   array_buffer[163].%X4;
			buf4.FinalHoldPosition.Enable._29 				        :=   array_buffer[163].%X5;
			buf4.FinalHoldPosition.Enable._30 				        :=   array_buffer[163].%X6;
			buf4.FinalHoldPosition.Enable._31 				        :=   array_buffer[163].%X7;
			buf4.FinalHoldPosition.LowerBad:=       TO_DINT(SHL(TO_DWORD(array_buffer[164]), UINT#24) OR
															SHL(TO_DWORD(array_buffer[165]), UINT#16) OR
															SHL(TO_DWORD(array_buffer[166]),  UINT#8) OR
																TO_DWORD(array_buffer[167]));
			buf4.FinalHoldPosition.LowerSuspect:=   TO_DINT(SHL(TO_DWORD(array_buffer[168]), UINT#24) OR
															SHL(TO_DWORD(array_buffer[169]), UINT#16) OR
															SHL(TO_DWORD(array_buffer[170]),  UINT#8) OR
																TO_DWORD(array_buffer[171]));
			buf4.FinalHoldPosition.UpperSuspect:=   TO_DINT(SHL(TO_DWORD(array_buffer[172]), UINT#24) OR
															SHL(TO_DWORD(array_buffer[173]), UINT#16) OR
															SHL(TO_DWORD(array_buffer[174]),  UINT#8) OR
																TO_DWORD(array_buffer[175]));
			buf4.FinalHoldPosition.UpperBad:=       TO_DINT(SHL(TO_DWORD(array_buffer[176]), UINT#24) OR
															SHL(TO_DWORD(array_buffer[177]), UINT#16) OR
															SHL(TO_DWORD(array_buffer[178]),  UINT#8) OR
																TO_DWORD(array_buffer[179]));
			buf4.ErrorStatus.Enable._0 				                :=   array_buffer[180].%X0;
			buf4.ErrorStatus.Enable._1 				                :=   array_buffer[180].%X1;
			buf4.ErrorStatus.Enable._2 				                :=   array_buffer[180].%X2;
			buf4.ErrorStatus.Enable._3 				                :=   array_buffer[180].%X3;
			buf4.ErrorStatus.Enable._4 				                :=   array_buffer[180].%X4;
			buf4.ErrorStatus.Enable._5 				                :=   array_buffer[180].%X5;
			buf4.ErrorStatus.Enable._6 				                :=   array_buffer[180].%X6;
			buf4.ErrorStatus.Enable._7 				                :=   array_buffer[180].%X7;
			buf4.ErrorStatus.Enable._8 				                :=   array_buffer[181].%X0;
			buf4.ErrorStatus.Enable._9 				                :=   array_buffer[181].%X1;
			buf4.ErrorStatus.Enable._10 				            :=   array_buffer[181].%X2;
			buf4.ErrorStatus.Enable._11 				            :=   array_buffer[181].%X3;
			buf4.ErrorStatus.Enable._12 				            :=   array_buffer[181].%X4;
			buf4.ErrorStatus.Enable._13 				            :=   array_buffer[181].%X5;
			buf4.ErrorStatus.Enable._14 				            :=   array_buffer[181].%X6;
			buf4.ErrorStatus.Enable._15 				            :=   array_buffer[181].%X7;
			buf4.ErrorStatus.Enable._16 				            :=   array_buffer[182].%X0;
			buf4.ErrorStatus.Enable._17 				            :=   array_buffer[182].%X1;
			buf4.ErrorStatus.Enable._18 				            :=   array_buffer[182].%X2;
			buf4.ErrorStatus.Enable._19 				            :=   array_buffer[182].%X3;
			buf4.ErrorStatus.Enable._20 				            :=   array_buffer[182].%X4;
			buf4.ErrorStatus.Enable._21 				            :=   array_buffer[182].%X5;
			buf4.ErrorStatus.Enable._22 				            :=   array_buffer[182].%X6;
			buf4.ErrorStatus.Enable._23 				            :=   array_buffer[182].%X7;
			buf4.ErrorStatus.Enable.LowerBad_1 		                :=   array_buffer[183].%X0;
			buf4.ErrorStatus.Enable.LowerSuspect_1 	                :=   array_buffer[183].%X1;
			buf4.ErrorStatus.Enable.UpperSuspect_1		            :=   array_buffer[183].%X2;
			buf4.ErrorStatus.Enable.UpperBad_1 		                :=   array_buffer[183].%X3;
			buf4.ErrorStatus.Enable.Display_1 			            :=   array_buffer[183].%X4;
			buf4.ErrorStatus.Enable._29 				            :=   array_buffer[183].%X5;
			buf4.ErrorStatus.Enable._30 				            :=   array_buffer[183].%X6;
			buf4.ErrorStatus.Enable._31 				            :=   array_buffer[183].%X7;
			buf4.ErrorStatus.LowerBad:=             TO_DINT(SHL(TO_DWORD(array_buffer[184]), UINT#24) OR
															SHL(TO_DWORD(array_buffer[185]), UINT#16) OR
															SHL(TO_DWORD(array_buffer[186]),  UINT#8) OR
																TO_DWORD(array_buffer[187]));
			buf4.ErrorStatus.LowerSuspect:=         TO_DINT(SHL(TO_DWORD(array_buffer[188]), UINT#24) OR
															SHL(TO_DWORD(array_buffer[189]), UINT#16) OR
															SHL(TO_DWORD(array_buffer[190]),  UINT#8) OR
																TO_DWORD(array_buffer[191]));
			buf4.ErrorStatus.UpperSuspect:=         TO_DINT(SHL(TO_DWORD(array_buffer[192]), UINT#24) OR
															SHL(TO_DWORD(array_buffer[193]), UINT#16) OR
															SHL(TO_DWORD(array_buffer[194]),  UINT#8) OR
																TO_DWORD(array_buffer[195]));
			buf4.ErrorStatus.UpperBad:=             TO_DINT(SHL(TO_DWORD(array_buffer[196]), UINT#24) OR
															SHL(TO_DWORD(array_buffer[197]), UINT#16) OR
															SHL(TO_DWORD(array_buffer[198]),  UINT#8) OR
																TO_DWORD(array_buffer[199]));
        END_METHOD

        METHOD PRIVATE ByteArray_TO_buf5
            VAR_INPUT
                array_buffer : ARRAY[0..253] OF BYTE;
            END_VAR
            VAR_IN_OUT
                buf5 : Axo_IQ_SeriesWelder_data5_176bytes;
            END_VAR
			buf5.AnalogSensor.Sensor[1].Enable:=    TO_DINT(SHL(TO_DWORD(array_buffer[  0]), UINT#24) OR
															SHL(TO_DWORD(array_buffer[  1]), UINT#16) OR
															SHL(TO_DWORD(array_buffer[  2]),  UINT#8) OR
																TO_DWORD(array_buffer[  3]));
			buf5.AnalogSensor.Sensor[1].MIN_VOLT:=  TO_DINT(SHL(TO_DWORD(array_buffer[  4]), UINT#24) OR
															SHL(TO_DWORD(array_buffer[  5]), UINT#16) OR
															SHL(TO_DWORD(array_buffer[  6]),  UINT#8) OR
																TO_DWORD(array_buffer[  7]));
			buf5.AnalogSensor.Sensor[1].MAX_VOLT:=  TO_DINT(SHL(TO_DWORD(array_buffer[  8]), UINT#24) OR
															SHL(TO_DWORD(array_buffer[  9]), UINT#16) OR
															SHL(TO_DWORD(array_buffer[ 10]),  UINT#8) OR
																TO_DWORD(array_buffer[ 11]));
			buf5.AnalogSensor.Sensor[1].MIN_VAL:=   TO_DINT(SHL(TO_DWORD(array_buffer[ 12]), UINT#24) OR
															SHL(TO_DWORD(array_buffer[ 13]), UINT#16) OR
															SHL(TO_DWORD(array_buffer[ 14]),  UINT#8) OR
																TO_DWORD(array_buffer[ 15]));
			buf5.AnalogSensor.Sensor[1].MAX_VAL:=   TO_DINT(SHL(TO_DWORD(array_buffer[ 16]), UINT#24) OR
															SHL(TO_DWORD(array_buffer[ 17]), UINT#16) OR
															SHL(TO_DWORD(array_buffer[ 18]),  UINT#8) OR
																TO_DWORD(array_buffer[ 19]));
			buf5.AnalogSensor.Sensor[2].Enable:=    TO_DINT(SHL(TO_DWORD(array_buffer[ 20]), UINT#24) OR
															SHL(TO_DWORD(array_buffer[ 21]), UINT#16) OR
															SHL(TO_DWORD(array_buffer[ 22]),  UINT#8) OR
																TO_DWORD(array_buffer[ 23]));
			buf5.AnalogSensor.Sensor[2].MIN_VOLT:=  TO_DINT(SHL(TO_DWORD(array_buffer[ 24]), UINT#24) OR
															SHL(TO_DWORD(array_buffer[ 25]), UINT#16) OR
															SHL(TO_DWORD(array_buffer[ 26]),  UINT#8) OR
																TO_DWORD(array_buffer[ 27]));
			buf5.AnalogSensor.Sensor[2].MAX_VOLT:=  TO_DINT(SHL(TO_DWORD(array_buffer[ 28]), UINT#24) OR
															SHL(TO_DWORD(array_buffer[ 29]), UINT#16) OR
															SHL(TO_DWORD(array_buffer[ 30]),  UINT#8) OR
																TO_DWORD(array_buffer[ 31]));
			buf5.AnalogSensor.Sensor[2].MIN_VAL:=   TO_DINT(SHL(TO_DWORD(array_buffer[ 32]), UINT#24) OR
															SHL(TO_DWORD(array_buffer[ 33]), UINT#16) OR
															SHL(TO_DWORD(array_buffer[ 34]),  UINT#8) OR
																TO_DWORD(array_buffer[ 35]));
			buf5.AnalogSensor.Sensor[2].MAX_VAL:=   TO_DINT(SHL(TO_DWORD(array_buffer[ 36]), UINT#24) OR
															SHL(TO_DWORD(array_buffer[ 37]), UINT#16) OR
															SHL(TO_DWORD(array_buffer[ 38]),  UINT#8) OR
																TO_DWORD(array_buffer[ 39]));
			buf5.AnalogSensor.Sensor[3].Enable:=    TO_DINT(SHL(TO_DWORD(array_buffer[ 40]), UINT#24) OR
															SHL(TO_DWORD(array_buffer[ 41]), UINT#16) OR
															SHL(TO_DWORD(array_buffer[ 42]),  UINT#8) OR
																TO_DWORD(array_buffer[ 43]));
			buf5.AnalogSensor.Sensor[3].MIN_VOLT:=  TO_DINT(SHL(TO_DWORD(array_buffer[ 44]), UINT#24) OR
															SHL(TO_DWORD(array_buffer[ 45]), UINT#16) OR
															SHL(TO_DWORD(array_buffer[ 46]),  UINT#8) OR
																TO_DWORD(array_buffer[ 47]));
			buf5.AnalogSensor.Sensor[3].MAX_VOLT:=  TO_DINT(SHL(TO_DWORD(array_buffer[ 48]), UINT#24) OR
															SHL(TO_DWORD(array_buffer[ 49]), UINT#16) OR
															SHL(TO_DWORD(array_buffer[ 50]),  UINT#8) OR
																TO_DWORD(array_buffer[ 51]));
			buf5.AnalogSensor.Sensor[3].MIN_VAL:=   TO_DINT(SHL(TO_DWORD(array_buffer[ 52]), UINT#24) OR
															SHL(TO_DWORD(array_buffer[ 53]), UINT#16) OR
															SHL(TO_DWORD(array_buffer[ 54]),  UINT#8) OR
																TO_DWORD(array_buffer[ 55]));
			buf5.AnalogSensor.Sensor[3].MAX_VAL:=   TO_DINT(SHL(TO_DWORD(array_buffer[ 56]), UINT#24) OR
															SHL(TO_DWORD(array_buffer[ 57]), UINT#16) OR
															SHL(TO_DWORD(array_buffer[ 58]),  UINT#8) OR
																TO_DWORD(array_buffer[ 59]));
			buf5.AnalogSensor.Sensor[4].Enable:=    TO_DINT(SHL(TO_DWORD(array_buffer[ 60]), UINT#24) OR
															SHL(TO_DWORD(array_buffer[ 61]), UINT#16) OR
															SHL(TO_DWORD(array_buffer[ 62]),  UINT#8) OR
																TO_DWORD(array_buffer[ 63]));
			buf5.AnalogSensor.Sensor[4].MIN_VOLT:=  TO_DINT(SHL(TO_DWORD(array_buffer[ 64]), UINT#24) OR
															SHL(TO_DWORD(array_buffer[ 65]), UINT#16) OR
															SHL(TO_DWORD(array_buffer[ 66]),  UINT#8) OR
																TO_DWORD(array_buffer[ 67]));
			buf5.AnalogSensor.Sensor[4].MAX_VOLT:=  TO_DINT(SHL(TO_DWORD(array_buffer[ 68]), UINT#24) OR
															SHL(TO_DWORD(array_buffer[ 69]), UINT#16) OR
															SHL(TO_DWORD(array_buffer[ 70]),  UINT#8) OR
																TO_DWORD(array_buffer[ 71]));
			buf5.AnalogSensor.Sensor[4].MIN_VAL:=   TO_DINT(SHL(TO_DWORD(array_buffer[ 72]), UINT#24) OR
															SHL(TO_DWORD(array_buffer[ 73]), UINT#16) OR
															SHL(TO_DWORD(array_buffer[ 74]),  UINT#8) OR
																TO_DWORD(array_buffer[ 75]));
			buf5.AnalogSensor.Sensor[4].MAX_VAL:=   TO_DINT(SHL(TO_DWORD(array_buffer[ 76]), UINT#24) OR
															SHL(TO_DWORD(array_buffer[ 77]), UINT#16) OR
															SHL(TO_DWORD(array_buffer[ 78]),  UINT#8) OR
																TO_DWORD(array_buffer[ 79]));
			buf5.AnalogSensor.Sensor[5].Enable:=    TO_DINT(SHL(TO_DWORD(array_buffer[ 80]), UINT#24) OR
															SHL(TO_DWORD(array_buffer[ 81]), UINT#16) OR
															SHL(TO_DWORD(array_buffer[ 82]),  UINT#8) OR
																TO_DWORD(array_buffer[ 83]));
			buf5.AnalogSensor.Sensor[5].MIN_VOLT:=  TO_DINT(SHL(TO_DWORD(array_buffer[ 84]), UINT#24) OR
															SHL(TO_DWORD(array_buffer[ 85]), UINT#16) OR
															SHL(TO_DWORD(array_buffer[ 86]),  UINT#8) OR
																TO_DWORD(array_buffer[ 87]));
			buf5.AnalogSensor.Sensor[5].MAX_VOLT:=  TO_DINT(SHL(TO_DWORD(array_buffer[ 88]), UINT#24) OR
															SHL(TO_DWORD(array_buffer[ 89]), UINT#16) OR
															SHL(TO_DWORD(array_buffer[ 90]),  UINT#8) OR
																TO_DWORD(array_buffer[ 91]));
			buf5.AnalogSensor.Sensor[5].MIN_VAL:=   TO_DINT(SHL(TO_DWORD(array_buffer[ 92]), UINT#24) OR
															SHL(TO_DWORD(array_buffer[ 93]), UINT#16) OR
															SHL(TO_DWORD(array_buffer[ 94]),  UINT#8) OR
																TO_DWORD(array_buffer[ 95]));
			buf5.AnalogSensor.Sensor[5].MAX_VAL:=   TO_DINT(SHL(TO_DWORD(array_buffer[ 96]), UINT#24) OR
															SHL(TO_DWORD(array_buffer[ 97]), UINT#16) OR
															SHL(TO_DWORD(array_buffer[ 98]),  UINT#8) OR
																TO_DWORD(array_buffer[ 99]));
			buf5.AnalogSensor.Sensor[6].Enable:=    TO_DINT(SHL(TO_DWORD(array_buffer[100]), UINT#24) OR
															SHL(TO_DWORD(array_buffer[101]), UINT#16) OR
															SHL(TO_DWORD(array_buffer[102]),  UINT#8) OR
																TO_DWORD(array_buffer[103]));
			buf5.AnalogSensor.Sensor[6].MIN_VOLT:=  TO_DINT(SHL(TO_DWORD(array_buffer[104]), UINT#24) OR
															SHL(TO_DWORD(array_buffer[105]), UINT#16) OR
															SHL(TO_DWORD(array_buffer[106]),  UINT#8) OR
																TO_DWORD(array_buffer[107]));
			buf5.AnalogSensor.Sensor[6].MAX_VOLT:=  TO_DINT(SHL(TO_DWORD(array_buffer[108]), UINT#24) OR
															SHL(TO_DWORD(array_buffer[109]), UINT#16) OR
															SHL(TO_DWORD(array_buffer[110]),  UINT#8) OR
																TO_DWORD(array_buffer[111]));
			buf5.AnalogSensor.Sensor[6].MIN_VAL:=   TO_DINT(SHL(TO_DWORD(array_buffer[112]), UINT#24) OR
															SHL(TO_DWORD(array_buffer[113]), UINT#16) OR
															SHL(TO_DWORD(array_buffer[114]),  UINT#8) OR
																TO_DWORD(array_buffer[115]));
			buf5.AnalogSensor.Sensor[6].MAX_VAL:=   TO_DINT(SHL(TO_DWORD(array_buffer[116]), UINT#24) OR
															SHL(TO_DWORD(array_buffer[117]), UINT#16) OR
															SHL(TO_DWORD(array_buffer[118]),  UINT#8) OR
																TO_DWORD(array_buffer[119]));
			buf5.AnalogSensor.Sensor[7].Enable:=    TO_DINT(SHL(TO_DWORD(array_buffer[120]), UINT#24) OR
															SHL(TO_DWORD(array_buffer[121]), UINT#16) OR
															SHL(TO_DWORD(array_buffer[122]),  UINT#8) OR
																TO_DWORD(array_buffer[123]));
			buf5.AnalogSensor.Sensor[7].MIN_VOLT:=  TO_DINT(SHL(TO_DWORD(array_buffer[124]), UINT#24) OR
															SHL(TO_DWORD(array_buffer[125]), UINT#16) OR
															SHL(TO_DWORD(array_buffer[126]),  UINT#8) OR
																TO_DWORD(array_buffer[127]));
			buf5.AnalogSensor.Sensor[7].MAX_VOLT:=  TO_DINT(SHL(TO_DWORD(array_buffer[128]), UINT#24) OR
															SHL(TO_DWORD(array_buffer[129]), UINT#16) OR
															SHL(TO_DWORD(array_buffer[130]),  UINT#8) OR
																TO_DWORD(array_buffer[131]));
			buf5.AnalogSensor.Sensor[7].MIN_VAL:=   TO_DINT(SHL(TO_DWORD(array_buffer[132]), UINT#24) OR
															SHL(TO_DWORD(array_buffer[133]), UINT#16) OR
															SHL(TO_DWORD(array_buffer[134]),  UINT#8) OR
																TO_DWORD(array_buffer[135]));
			buf5.AnalogSensor.Sensor[7].MAX_VAL:=   TO_DINT(SHL(TO_DWORD(array_buffer[136]), UINT#24) OR
															SHL(TO_DWORD(array_buffer[137]), UINT#16) OR
															SHL(TO_DWORD(array_buffer[138]),  UINT#8) OR
																TO_DWORD(array_buffer[139]));
			buf5.AnalogSensor.Sensor[8].Enable:=    TO_DINT(SHL(TO_DWORD(array_buffer[140]), UINT#24) OR
															SHL(TO_DWORD(array_buffer[141]), UINT#16) OR
															SHL(TO_DWORD(array_buffer[142]),  UINT#8) OR
																TO_DWORD(array_buffer[143]));
			buf5.AnalogSensor.Sensor[8].MIN_VOLT:=  TO_DINT(SHL(TO_DWORD(array_buffer[144]), UINT#24) OR
															SHL(TO_DWORD(array_buffer[145]), UINT#16) OR
															SHL(TO_DWORD(array_buffer[146]),  UINT#8) OR
																TO_DWORD(array_buffer[147]));
			buf5.AnalogSensor.Sensor[8].MAX_VOLT:=  TO_DINT(SHL(TO_DWORD(array_buffer[148]), UINT#24) OR
															SHL(TO_DWORD(array_buffer[149]), UINT#16) OR
															SHL(TO_DWORD(array_buffer[150]),  UINT#8) OR
																TO_DWORD(array_buffer[151]));
			buf5.AnalogSensor.Sensor[8].MIN_VAL:=   TO_DINT(SHL(TO_DWORD(array_buffer[152]), UINT#24) OR
															SHL(TO_DWORD(array_buffer[153]), UINT#16) OR
															SHL(TO_DWORD(array_buffer[154]),  UINT#8) OR
																TO_DWORD(array_buffer[155]));
			buf5.AnalogSensor.Sensor[8].MAX_VAL:=   TO_DINT(SHL(TO_DWORD(array_buffer[156]), UINT#24) OR
															SHL(TO_DWORD(array_buffer[157]), UINT#16) OR
															SHL(TO_DWORD(array_buffer[158]),  UINT#8) OR
																TO_DWORD(array_buffer[159]));
			buf5.AfterburstEnable:=                 TO_DINT(SHL(TO_DWORD(array_buffer[160]), UINT#24) OR
															SHL(TO_DWORD(array_buffer[161]), UINT#16) OR
															SHL(TO_DWORD(array_buffer[162]),  UINT#8) OR
																TO_DWORD(array_buffer[163]));
			buf5.LimitWeld1TimeEnable._0 				:=               array_buffer[164].%X0;
			buf5.LimitWeld1TimeEnable._1 				:=               array_buffer[164].%X1;
			buf5.LimitWeld1TimeEnable._2 				:=               array_buffer[164].%X2;
			buf5.LimitWeld1TimeEnable._3 				:=               array_buffer[164].%X3;
			buf5.LimitWeld1TimeEnable._4 				:=               array_buffer[164].%X4;
			buf5.LimitWeld1TimeEnable._5 				:=               array_buffer[164].%X5;
			buf5.LimitWeld1TimeEnable._6 				:=               array_buffer[164].%X6;
			buf5.LimitWeld1TimeEnable._7 				:=               array_buffer[164].%X7;
			buf5.LimitWeld1TimeEnable._8 				:=               array_buffer[165].%X0;
			buf5.LimitWeld1TimeEnable._9 				:=               array_buffer[165].%X1;
			buf5.LimitWeld1TimeEnable._10 				:=               array_buffer[165].%X2;
			buf5.LimitWeld1TimeEnable._11 				:=               array_buffer[165].%X3;
			buf5.LimitWeld1TimeEnable._12 				:=               array_buffer[165].%X4;
			buf5.LimitWeld1TimeEnable._13 				:=               array_buffer[165].%X5;
			buf5.LimitWeld1TimeEnable._14 				:=               array_buffer[165].%X6;
			buf5.LimitWeld1TimeEnable._15 				:=               array_buffer[165].%X7;
			buf5.LimitWeld1TimeEnable._16 				:=               array_buffer[166].%X0;
			buf5.LimitWeld1TimeEnable._17 				:=               array_buffer[166].%X1;
			buf5.LimitWeld1TimeEnable._18 				:=               array_buffer[166].%X2;
			buf5.LimitWeld1TimeEnable._19 				:=               array_buffer[166].%X3;
			buf5.LimitWeld1TimeEnable._20 				:=               array_buffer[166].%X4;
			buf5.LimitWeld1TimeEnable._21 				:=               array_buffer[166].%X5;
			buf5.LimitWeld1TimeEnable._22 				:=               array_buffer[166].%X6;
			buf5.LimitWeld1TimeEnable._23 				:=               array_buffer[166].%X7;
			buf5.LimitWeld1TimeEnable.LowerBad_1 		:=               array_buffer[167].%X0;
			buf5.LimitWeld1TimeEnable.LowerSuspect_1	:=               array_buffer[167].%X1;
			buf5.LimitWeld1TimeEnable.UpperSuspect_1	:=               array_buffer[167].%X2;
			buf5.LimitWeld1TimeEnable.UpperBad_1 		:=               array_buffer[167].%X3;
			buf5.LimitWeld1TimeEnable.Display_1 		:=               array_buffer[167].%X4;
			buf5.LimitWeld1TimeEnable._29 				:=               array_buffer[167].%X5;
			buf5.LimitWeld1TimeEnable._30 				:=               array_buffer[167].%X6;
			buf5.LimitWeld1TimeEnable._31 				:=               array_buffer[167].%X7;
			buf5.LimitWeld1EnergyEnable._0 				:=               array_buffer[168].%X0;
			buf5.LimitWeld1EnergyEnable._1 				:=               array_buffer[168].%X1;
			buf5.LimitWeld1EnergyEnable._2 				:=               array_buffer[168].%X2;
			buf5.LimitWeld1EnergyEnable._3 				:=               array_buffer[168].%X3;
			buf5.LimitWeld1EnergyEnable._4 				:=               array_buffer[168].%X4;
			buf5.LimitWeld1EnergyEnable._5 				:=               array_buffer[168].%X5;
			buf5.LimitWeld1EnergyEnable._6 				:=               array_buffer[168].%X6;
			buf5.LimitWeld1EnergyEnable._7 				:=               array_buffer[168].%X7;
			buf5.LimitWeld1EnergyEnable._8 				:=               array_buffer[169].%X0;
			buf5.LimitWeld1EnergyEnable._9 				:=               array_buffer[169].%X1;
			buf5.LimitWeld1EnergyEnable._10 		    :=               array_buffer[169].%X2;
			buf5.LimitWeld1EnergyEnable._11 		    :=               array_buffer[169].%X3;
			buf5.LimitWeld1EnergyEnable._12 		    :=               array_buffer[169].%X4;
			buf5.LimitWeld1EnergyEnable._13 		    :=               array_buffer[169].%X5;
			buf5.LimitWeld1EnergyEnable._14 		    :=               array_buffer[169].%X6;
			buf5.LimitWeld1EnergyEnable._15 		    :=               array_buffer[169].%X7;
			buf5.LimitWeld1EnergyEnable._16 		    :=               array_buffer[170].%X0;
			buf5.LimitWeld1EnergyEnable._17 		    :=               array_buffer[170].%X1;
			buf5.LimitWeld1EnergyEnable._18 		    :=               array_buffer[170].%X2;
			buf5.LimitWeld1EnergyEnable._19 		    :=               array_buffer[170].%X3;
			buf5.LimitWeld1EnergyEnable._20 		    :=               array_buffer[170].%X4;
			buf5.LimitWeld1EnergyEnable._21 		    :=               array_buffer[170].%X5;
			buf5.LimitWeld1EnergyEnable._22 		    :=               array_buffer[170].%X6;
			buf5.LimitWeld1EnergyEnable._23 		    :=               array_buffer[170].%X7;
			buf5.LimitWeld1EnergyEnable.LowerBad_1 		:=               array_buffer[171].%X0;
			buf5.LimitWeld1EnergyEnable.LowerSuspect_1	:=               array_buffer[171].%X1;
			buf5.LimitWeld1EnergyEnable.UpperSuspect_1	:=               array_buffer[171].%X2;
			buf5.LimitWeld1EnergyEnable.UpperBad_1 		:=               array_buffer[171].%X3;
			buf5.LimitWeld1EnergyEnable.Display_1 		:=               array_buffer[171].%X4;
			buf5.LimitWeld1EnergyEnable._29 			:=               array_buffer[171].%X5;
			buf5.LimitWeld1EnergyEnable._30 			:=               array_buffer[171].%X6;
			buf5.LimitWeld1EnergyEnable._31 			:=               array_buffer[171].%X7;
			buf5.LimitWeld1PowerEnable._0 				:=               array_buffer[172].%X0;
			buf5.LimitWeld1PowerEnable._1 				:=               array_buffer[172].%X1;
			buf5.LimitWeld1PowerEnable._2 				:=               array_buffer[172].%X2;
			buf5.LimitWeld1PowerEnable._3 				:=               array_buffer[172].%X3;
			buf5.LimitWeld1PowerEnable._4 				:=               array_buffer[172].%X4;
			buf5.LimitWeld1PowerEnable._5 				:=               array_buffer[172].%X5;
			buf5.LimitWeld1PowerEnable._6 				:=               array_buffer[172].%X6;
			buf5.LimitWeld1PowerEnable._7 				:=               array_buffer[172].%X7;
			buf5.LimitWeld1PowerEnable._8 				:=               array_buffer[173].%X0;
			buf5.LimitWeld1PowerEnable._9 				:=               array_buffer[173].%X1;
			buf5.LimitWeld1PowerEnable._10 				:=               array_buffer[173].%X2;
			buf5.LimitWeld1PowerEnable._11 				:=               array_buffer[173].%X3;
			buf5.LimitWeld1PowerEnable._12 				:=               array_buffer[173].%X4;
			buf5.LimitWeld1PowerEnable._13 				:=               array_buffer[173].%X5;
			buf5.LimitWeld1PowerEnable._14 				:=               array_buffer[173].%X6;
			buf5.LimitWeld1PowerEnable._15 				:=               array_buffer[173].%X7;
			buf5.LimitWeld1PowerEnable._16 				:=               array_buffer[174].%X0;
			buf5.LimitWeld1PowerEnable._17 				:=               array_buffer[174].%X1;
			buf5.LimitWeld1PowerEnable._18 				:=               array_buffer[174].%X2;
			buf5.LimitWeld1PowerEnable._19 				:=               array_buffer[174].%X3;
			buf5.LimitWeld1PowerEnable._20 				:=               array_buffer[174].%X4;
			buf5.LimitWeld1PowerEnable._21 				:=               array_buffer[174].%X5;
			buf5.LimitWeld1PowerEnable._22 				:=               array_buffer[174].%X6;
			buf5.LimitWeld1PowerEnable._23 				:=               array_buffer[174].%X7;
			buf5.LimitWeld1PowerEnable.LowerBad_1 		:=               array_buffer[175].%X0;
			buf5.LimitWeld1PowerEnable.LowerSuspect_1	:=               array_buffer[175].%X1;
			buf5.LimitWeld1PowerEnable.UpperSuspect_1	:=               array_buffer[175].%X2;
			buf5.LimitWeld1PowerEnable.UpperBad_1 		:=               array_buffer[175].%X3;
			buf5.LimitWeld1PowerEnable.Display_1 		:=               array_buffer[175].%X4;
			buf5.LimitWeld1PowerEnable._29 				:=               array_buffer[175].%X5;
			buf5.LimitWeld1PowerEnable._30 				:=               array_buffer[175].%X6;
			buf5.LimitWeld1PowerEnable._31 				:=               array_buffer[175].%X7;
		END_METHOD

        METHOD PRIVATE buf1_TO_ByteArray
            VAR_IN_OUT
                buf1 : Axo_IQ_SeriesWelder_data1_132bytes;
                array_buffer : ARRAY[0..253] OF BYTE;
            END_VAR

            // ---- ProcCtrl: DINT fields → bytes ----
            array_buffer[  0] := TO_BYTE(SHR(TO_DWORD(buf1.ProcCtrl.RegulationAmplitude), UINT#24));
            array_buffer[  1] := TO_BYTE(SHR(TO_DWORD(buf1.ProcCtrl.RegulationAmplitude), UINT#16));
            array_buffer[  2] := TO_BYTE(SHR(TO_DWORD(buf1.ProcCtrl.RegulationAmplitude),  UINT#8));
            array_buffer[  3] := TO_BYTE(     TO_DWORD(buf1.ProcCtrl.RegulationAmplitude));

            array_buffer[  4] := TO_BYTE(SHR(TO_DWORD(buf1.ProcCtrl.RampUpTime), UINT#24));
            array_buffer[  5] := TO_BYTE(SHR(TO_DWORD(buf1.ProcCtrl.RampUpTime), UINT#16));
            array_buffer[  6] := TO_BYTE(SHR(TO_DWORD(buf1.ProcCtrl.RampUpTime),  UINT#8));
            array_buffer[  7] := TO_BYTE(     TO_DWORD(buf1.ProcCtrl.RampUpTime));

            array_buffer[  8] := TO_BYTE(SHR(TO_DWORD(buf1.ProcCtrl.RampDownTime), UINT#24));
            array_buffer[  9] := TO_BYTE(SHR(TO_DWORD(buf1.ProcCtrl.RampDownTime), UINT#16));
            array_buffer[ 10] := TO_BYTE(SHR(TO_DWORD(buf1.ProcCtrl.RampDownTime),  UINT#8));
            array_buffer[ 11] := TO_BYTE(     TO_DWORD(buf1.ProcCtrl.RampDownTime));

            // ---- ProcCtrl: OBSOLETE_ProcessControlEnable bits → bytes 12..15 ----
            array_buffer[12].%X0 := buf1.ProcCtrl.OBSOLETE_ProcessControlEnable._0;
            array_buffer[12].%X1 := buf1.ProcCtrl.OBSOLETE_ProcessControlEnable._1;
            array_buffer[12].%X2 := buf1.ProcCtrl.OBSOLETE_ProcessControlEnable._2;
            array_buffer[12].%X3 := buf1.ProcCtrl.OBSOLETE_ProcessControlEnable._3;
            array_buffer[12].%X4 := buf1.ProcCtrl.OBSOLETE_ProcessControlEnable._4;
            array_buffer[12].%X5 := buf1.ProcCtrl.OBSOLETE_ProcessControlEnable._5;
            array_buffer[12].%X6 := buf1.ProcCtrl.OBSOLETE_ProcessControlEnable._6;
            array_buffer[12].%X7 := buf1.ProcCtrl.OBSOLETE_ProcessControlEnable._7;

            array_buffer[13].%X0 := buf1.ProcCtrl.OBSOLETE_ProcessControlEnable.HoldTime_Enable;
            array_buffer[13].%X1 := buf1.ProcCtrl.OBSOLETE_ProcessControlEnable.Afterburst_Enable;
            array_buffer[13].%X2 := buf1.ProcCtrl.OBSOLETE_ProcessControlEnable._10;
            array_buffer[13].%X3 := buf1.ProcCtrl.OBSOLETE_ProcessControlEnable._11;
            array_buffer[13].%X4 := buf1.ProcCtrl.OBSOLETE_ProcessControlEnable._12;
            array_buffer[13].%X5 := buf1.ProcCtrl.OBSOLETE_ProcessControlEnable._13;
            array_buffer[13].%X6 := buf1.ProcCtrl.OBSOLETE_ProcessControlEnable._14;
            array_buffer[13].%X7 := buf1.ProcCtrl.OBSOLETE_ProcessControlEnable._15;

            array_buffer[14].%X0 := buf1.ProcCtrl.OBSOLETE_ProcessControlEnable._16;
            array_buffer[14].%X1 := buf1.ProcCtrl.OBSOLETE_ProcessControlEnable._17;
            array_buffer[14].%X2 := buf1.ProcCtrl.OBSOLETE_ProcessControlEnable._18;
            array_buffer[14].%X3 := buf1.ProcCtrl.OBSOLETE_ProcessControlEnable._19;
            array_buffer[14].%X4 := buf1.ProcCtrl.OBSOLETE_ProcessControlEnable._20;
            array_buffer[14].%X5 := buf1.ProcCtrl.OBSOLETE_ProcessControlEnable._21;
            array_buffer[14].%X6 := buf1.ProcCtrl.OBSOLETE_ProcessControlEnable._22;
            array_buffer[14].%X7 := buf1.ProcCtrl.OBSOLETE_ProcessControlEnable._23;

            array_buffer[15].%X0 := buf1.ProcCtrl.OBSOLETE_ProcessControlEnable.WeldTime_Enable;
            array_buffer[15].%X1 := buf1.ProcCtrl.OBSOLETE_ProcessControlEnable.WeldPower_Enable;
            array_buffer[15].%X2 := buf1.ProcCtrl.OBSOLETE_ProcessControlEnable.WeldEnergy_Enable;
            array_buffer[15].%X3 := buf1.ProcCtrl.OBSOLETE_ProcessControlEnable.WeldDistance_Enable;
            array_buffer[15].%X4 := buf1.ProcCtrl.OBSOLETE_ProcessControlEnable.WeldPosition_Enable;
            array_buffer[15].%X5 := buf1.ProcCtrl.OBSOLETE_ProcessControlEnable._29;
            array_buffer[15].%X6 := buf1.ProcCtrl.OBSOLETE_ProcessControlEnable._30;
            array_buffer[15].%X7 := buf1.ProcCtrl.OBSOLETE_ProcessControlEnable._31;

            // ---- ProcCtrl: more DINTs ----
            array_buffer[16] := TO_BYTE(SHR(TO_DWORD(buf1.ProcCtrl.WeldTime), UINT#24));
            array_buffer[17] := TO_BYTE(SHR(TO_DWORD(buf1.ProcCtrl.WeldTime), UINT#16));
            array_buffer[18] := TO_BYTE(SHR(TO_DWORD(buf1.ProcCtrl.WeldTime),  UINT#8));
            array_buffer[19] := TO_BYTE(     TO_DWORD(buf1.ProcCtrl.WeldTime));

            array_buffer[20] := TO_BYTE(SHR(TO_DWORD(buf1.ProcCtrl.WeldPower), UINT#24));
            array_buffer[21] := TO_BYTE(SHR(TO_DWORD(buf1.ProcCtrl.WeldPower), UINT#16));
            array_buffer[22] := TO_BYTE(SHR(TO_DWORD(buf1.ProcCtrl.WeldPower),  UINT#8));
            array_buffer[23] := TO_BYTE(     TO_DWORD(buf1.ProcCtrl.WeldPower));

            array_buffer[24] := TO_BYTE(SHR(TO_DWORD(buf1.ProcCtrl.WeldEnergy), UINT#24));
            array_buffer[25] := TO_BYTE(SHR(TO_DWORD(buf1.ProcCtrl.WeldEnergy), UINT#16));
            array_buffer[26] := TO_BYTE(SHR(TO_DWORD(buf1.ProcCtrl.WeldEnergy),  UINT#8));
            array_buffer[27] := TO_BYTE(     TO_DWORD(buf1.ProcCtrl.WeldEnergy));

            array_buffer[28] := TO_BYTE(SHR(TO_DWORD(buf1.ProcCtrl.HoldTime), UINT#24));
            array_buffer[29] := TO_BYTE(SHR(TO_DWORD(buf1.ProcCtrl.HoldTime), UINT#16));
            array_buffer[30] := TO_BYTE(SHR(TO_DWORD(buf1.ProcCtrl.HoldTime),  UINT#8));
            array_buffer[31] := TO_BYTE(     TO_DWORD(buf1.ProcCtrl.HoldTime));

            array_buffer[32] := TO_BYTE(SHR(TO_DWORD(buf1.ProcCtrl.AfterBurstDelay), UINT#24));
            array_buffer[33] := TO_BYTE(SHR(TO_DWORD(buf1.ProcCtrl.AfterBurstDelay), UINT#16));
            array_buffer[34] := TO_BYTE(SHR(TO_DWORD(buf1.ProcCtrl.AfterBurstDelay),  UINT#8));
            array_buffer[35] := TO_BYTE(     TO_DWORD(buf1.ProcCtrl.AfterBurstDelay));

            array_buffer[36] := TO_BYTE(SHR(TO_DWORD(buf1.ProcCtrl.AfterBurstDuration), UINT#24));
            array_buffer[37] := TO_BYTE(SHR(TO_DWORD(buf1.ProcCtrl.AfterBurstDuration), UINT#16));
            array_buffer[38] := TO_BYTE(SHR(TO_DWORD(buf1.ProcCtrl.AfterBurstDuration),  UINT#8));
            array_buffer[39] := TO_BYTE(     TO_DWORD(buf1.ProcCtrl.AfterBurstDuration));

            // ---- ProcLimits.Enable bits → bytes 40..43 ----
            array_buffer[40].%X0 := buf1.ProcLimits.Enable.LowerBadEnergy;
            array_buffer[40].%X1 := buf1.ProcLimits.Enable.LowerSuspectEnergy;
            array_buffer[40].%X2 := buf1.ProcLimits.Enable.UpperSuspectEnergy;
            array_buffer[40].%X3 := buf1.ProcLimits.Enable.UpperBadEnergy;
            array_buffer[40].%X4 := buf1.ProcLimits.Enable.DisplayEnergy;
            array_buffer[40].%X5 := buf1.ProcLimits.Enable._5;
            array_buffer[40].%X6 := buf1.ProcLimits.Enable._6;
            array_buffer[40].%X7 := buf1.ProcLimits.Enable._7;

            array_buffer[41].%X0 := buf1.ProcLimits.Enable.LowerBadPower;
            array_buffer[41].%X1 := buf1.ProcLimits.Enable.LowerSuspectPower;
            array_buffer[41].%X2 := buf1.ProcLimits.Enable.UpperSuspectPower;
            array_buffer[41].%X3 := buf1.ProcLimits.Enable.UpperBadPower;
            array_buffer[41].%X4 := buf1.ProcLimits.Enable.DisplayPower;
            array_buffer[41].%X5 := buf1.ProcLimits.Enable._13;
            array_buffer[41].%X6 := buf1.ProcLimits.Enable._14;
            array_buffer[41].%X7 := buf1.ProcLimits.Enable._15;

            array_buffer[42].%X0 := buf1.ProcLimits.Enable.LowerBadTime;
            array_buffer[42].%X1 := buf1.ProcLimits.Enable.LowerSuspectTime;
            array_buffer[42].%X2 := buf1.ProcLimits.Enable.UpperSuspectTime;
            array_buffer[42].%X3 := buf1.ProcLimits.Enable.UpperBadTIme; // note: name as in source
            array_buffer[42].%X4 := buf1.ProcLimits.Enable.DisplayTime;
            array_buffer[42].%X5 := buf1.ProcLimits.Enable._21;
            array_buffer[42].%X6 := buf1.ProcLimits.Enable._22;
            array_buffer[42].%X7 := buf1.ProcLimits.Enable._23;

            array_buffer[43].%X0 := buf1.ProcLimits.Enable._24;
            array_buffer[43].%X1 := buf1.ProcLimits.Enable._25;
            array_buffer[43].%X2 := buf1.ProcLimits.Enable._26;
            array_buffer[43].%X3 := buf1.ProcLimits.Enable._27;
            array_buffer[43].%X4 := buf1.ProcLimits.Enable._28;
            array_buffer[43].%X5 := buf1.ProcLimits.Enable._29;
            array_buffer[43].%X6 := buf1.ProcLimits.Enable._30;
            array_buffer[43].%X7 := buf1.ProcLimits.Enable._31;

            // ---- ProcLimits: DINTs ----
            array_buffer[44] := TO_BYTE(SHR(TO_DWORD(buf1.ProcLimits.WeldTimeLowerBad), UINT#24));
            array_buffer[45] := TO_BYTE(SHR(TO_DWORD(buf1.ProcLimits.WeldTimeLowerBad), UINT#16));
            array_buffer[46] := TO_BYTE(SHR(TO_DWORD(buf1.ProcLimits.WeldTimeLowerBad),  UINT#8));
            array_buffer[47] := TO_BYTE(     TO_DWORD(buf1.ProcLimits.WeldTimeLowerBad));

            array_buffer[48] := TO_BYTE(SHR(TO_DWORD(buf1.ProcLimits.WeldTimeLowerSuspect), UINT#24));
            array_buffer[49] := TO_BYTE(SHR(TO_DWORD(buf1.ProcLimits.WeldTimeLowerSuspect), UINT#16));
            array_buffer[50] := TO_BYTE(SHR(TO_DWORD(buf1.ProcLimits.WeldTimeLowerSuspect),  UINT#8));
            array_buffer[51] := TO_BYTE(     TO_DWORD(buf1.ProcLimits.WeldTimeLowerSuspect));

            array_buffer[52] := TO_BYTE(SHR(TO_DWORD(buf1.ProcLimits.WeldTimeUpperSuspect), UINT#24));
            array_buffer[53] := TO_BYTE(SHR(TO_DWORD(buf1.ProcLimits.WeldTimeUpperSuspect), UINT#16));
            array_buffer[54] := TO_BYTE(SHR(TO_DWORD(buf1.ProcLimits.WeldTimeUpperSuspect),  UINT#8));
            array_buffer[55] := TO_BYTE(     TO_DWORD(buf1.ProcLimits.WeldTimeUpperSuspect));

            array_buffer[56] := TO_BYTE(SHR(TO_DWORD(buf1.ProcLimits.WeldTimeUpperBad), UINT#24));
            array_buffer[57] := TO_BYTE(SHR(TO_DWORD(buf1.ProcLimits.WeldTimeUpperBad), UINT#16));
            array_buffer[58] := TO_BYTE(SHR(TO_DWORD(buf1.ProcLimits.WeldTimeUpperBad),  UINT#8));
            array_buffer[59] := TO_BYTE(     TO_DWORD(buf1.ProcLimits.WeldTimeUpperBad));

            array_buffer[60] := TO_BYTE(SHR(TO_DWORD(buf1.ProcLimits.WeldPowerLowerBad), UINT#24));
            array_buffer[61] := TO_BYTE(SHR(TO_DWORD(buf1.ProcLimits.WeldPowerLowerBad), UINT#16));
            array_buffer[62] := TO_BYTE(SHR(TO_DWORD(buf1.ProcLimits.WeldPowerLowerBad),  UINT#8));
            array_buffer[63] := TO_BYTE(     TO_DWORD(buf1.ProcLimits.WeldPowerLowerBad));

            array_buffer[64] := TO_BYTE(SHR(TO_DWORD(buf1.ProcLimits.WeldPwrLowerSuspect), UINT#24));
            array_buffer[65] := TO_BYTE(SHR(TO_DWORD(buf1.ProcLimits.WeldPwrLowerSuspect), UINT#16));
            array_buffer[66] := TO_BYTE(SHR(TO_DWORD(buf1.ProcLimits.WeldPwrLowerSuspect),  UINT#8));
            array_buffer[67] := TO_BYTE(     TO_DWORD(buf1.ProcLimits.WeldPwrLowerSuspect));

            array_buffer[68] := TO_BYTE(SHR(TO_DWORD(buf1.ProcLimits.WeldPwrUpperSuspect), UINT#24));
            array_buffer[69] := TO_BYTE(SHR(TO_DWORD(buf1.ProcLimits.WeldPwrUpperSuspect), UINT#16));
            array_buffer[70] := TO_BYTE(SHR(TO_DWORD(buf1.ProcLimits.WeldPwrUpperSuspect),  UINT#8));
            array_buffer[71] := TO_BYTE(     TO_DWORD(buf1.ProcLimits.WeldPwrUpperSuspect));

            array_buffer[72] := TO_BYTE(SHR(TO_DWORD(buf1.ProcLimits.WeldPowerUpperBad), UINT#24));
            array_buffer[73] := TO_BYTE(SHR(TO_DWORD(buf1.ProcLimits.WeldPowerUpperBad), UINT#16));
            array_buffer[74] := TO_BYTE(SHR(TO_DWORD(buf1.ProcLimits.WeldPowerUpperBad),  UINT#8));
            array_buffer[75] := TO_BYTE(     TO_DWORD(buf1.ProcLimits.WeldPowerUpperBad));

            array_buffer[76] := TO_BYTE(SHR(TO_DWORD(buf1.ProcLimits.WeldEnergyLowerBad), UINT#24));
            array_buffer[77] := TO_BYTE(SHR(TO_DWORD(buf1.ProcLimits.WeldEnergyLowerBad), UINT#16));
            array_buffer[78] := TO_BYTE(SHR(TO_DWORD(buf1.ProcLimits.WeldEnergyLowerBad),  UINT#8));
            array_buffer[79] := TO_BYTE(     TO_DWORD(buf1.ProcLimits.WeldEnergyLowerBad));

            array_buffer[80] := TO_BYTE(SHR(TO_DWORD(buf1.ProcLimits.WeldEnergyLowerSuspect), UINT#24));
            array_buffer[81] := TO_BYTE(SHR(TO_DWORD(buf1.ProcLimits.WeldEnergyLowerSuspect), UINT#16));
            array_buffer[82] := TO_BYTE(SHR(TO_DWORD(buf1.ProcLimits.WeldEnergyLowerSuspect),  UINT#8));
            array_buffer[83] := TO_BYTE(     TO_DWORD(buf1.ProcLimits.WeldEnergyLowerSuspect));

            array_buffer[84] := TO_BYTE(SHR(TO_DWORD(buf1.ProcLimits.WeldEnergyUpperSuspect), UINT#24));
            array_buffer[85] := TO_BYTE(SHR(TO_DWORD(buf1.ProcLimits.WeldEnergyUpperSuspect), UINT#16));
            array_buffer[86] := TO_BYTE(SHR(TO_DWORD(buf1.ProcLimits.WeldEnergyUpperSuspect),  UINT#8));
            array_buffer[87] := TO_BYTE(     TO_DWORD(buf1.ProcLimits.WeldEnergyUpperSuspect));

            array_buffer[88] := TO_BYTE(SHR(TO_DWORD(buf1.ProcLimits.WeldEnergyUpperBad), UINT#24));
            array_buffer[89] := TO_BYTE(SHR(TO_DWORD(buf1.ProcLimits.WeldEnergyUpperBad), UINT#16));
            array_buffer[90] := TO_BYTE(SHR(TO_DWORD(buf1.ProcLimits.WeldEnergyUpperBad),  UINT#8));
            array_buffer[91] := TO_BYTE(     TO_DWORD(buf1.ProcLimits.WeldEnergyUpperBad));

            // ---- FreqCtrl: DINTs ----
            array_buffer[92] := TO_BYTE(SHR(TO_DWORD(buf1.FreqCtrl.FreerunFrequency), UINT#24));
            array_buffer[93] := TO_BYTE(SHR(TO_DWORD(buf1.FreqCtrl.FreerunFrequency), UINT#16));
            array_buffer[94] := TO_BYTE(SHR(TO_DWORD(buf1.FreqCtrl.FreerunFrequency),  UINT#8));
            array_buffer[95] := TO_BYTE(     TO_DWORD(buf1.FreqCtrl.FreerunFrequency));

            array_buffer[96] := TO_BYTE(SHR(TO_DWORD(buf1.FreqCtrl.LowerFrequencyBound), UINT#24));
            array_buffer[97] := TO_BYTE(SHR(TO_DWORD(buf1.FreqCtrl.LowerFrequencyBound), UINT#16));
            array_buffer[98] := TO_BYTE(SHR(TO_DWORD(buf1.FreqCtrl.LowerFrequencyBound),  UINT#8));
            array_buffer[99] := TO_BYTE(     TO_DWORD(buf1.FreqCtrl.LowerFrequencyBound));

            array_buffer[100] := TO_BYTE(SHR(TO_DWORD(buf1.FreqCtrl.UpperFrequencyBound), UINT#24));
            array_buffer[101] := TO_BYTE(SHR(TO_DWORD(buf1.FreqCtrl.UpperFrequencyBound), UINT#16));
            array_buffer[102] := TO_BYTE(SHR(TO_DWORD(buf1.FreqCtrl.UpperFrequencyBound),  UINT#8));
            array_buffer[103] := TO_BYTE(     TO_DWORD(buf1.FreqCtrl.UpperFrequencyBound));

            array_buffer[104] := TO_BYTE(SHR(TO_DWORD(buf1.FreqCtrl.LockandHoldModeEnable), UINT#24));
            array_buffer[105] := TO_BYTE(SHR(TO_DWORD(buf1.FreqCtrl.LockandHoldModeEnable), UINT#16));
            array_buffer[106] := TO_BYTE(SHR(TO_DWORD(buf1.FreqCtrl.LockandHoldModeEnable),  UINT#8));
            array_buffer[107] := TO_BYTE(     TO_DWORD(buf1.FreqCtrl.LockandHoldModeEnable));

            array_buffer[108] := TO_BYTE(SHR(TO_DWORD(buf1.FreqCtrl.USPhaseAdjustment), UINT#24));
            array_buffer[109] := TO_BYTE(SHR(TO_DWORD(buf1.FreqCtrl.USPhaseAdjustment), UINT#16));
            array_buffer[110] := TO_BYTE(SHR(TO_DWORD(buf1.FreqCtrl.USPhaseAdjustment),  UINT#8));
            array_buffer[111] := TO_BYTE(     TO_DWORD(buf1.FreqCtrl.USPhaseAdjustment));

            // ---- TriggerByPower: DINTs ----
            array_buffer[112] := TO_BYTE(SHR(TO_DWORD(buf1.TriggerByPower.Enable), UINT#24));
            array_buffer[113] := TO_BYTE(SHR(TO_DWORD(buf1.TriggerByPower.Enable), UINT#16));
            array_buffer[114] := TO_BYTE(SHR(TO_DWORD(buf1.TriggerByPower.Enable),  UINT#8));
            array_buffer[115] := TO_BYTE(     TO_DWORD(buf1.TriggerByPower.Enable));

            array_buffer[116] := TO_BYTE(SHR(TO_DWORD(buf1.TriggerByPower.Trigger_Timout), UINT#24));
            array_buffer[117] := TO_BYTE(SHR(TO_DWORD(buf1.TriggerByPower.Trigger_Timout), UINT#16));
            array_buffer[118] := TO_BYTE(SHR(TO_DWORD(buf1.TriggerByPower.Trigger_Timout),  UINT#8));
            array_buffer[119] := TO_BYTE(     TO_DWORD(buf1.TriggerByPower.Trigger_Timout));

            array_buffer[120] := TO_BYTE(SHR(TO_DWORD(buf1.TriggerByPower.Trigger_Level), UINT#24));
            array_buffer[121] := TO_BYTE(SHR(TO_DWORD(buf1.TriggerByPower.Trigger_Level), UINT#16));
            array_buffer[122] := TO_BYTE(SHR(TO_DWORD(buf1.TriggerByPower.Trigger_Level),  UINT#8));
            array_buffer[123] := TO_BYTE(     TO_DWORD(buf1.TriggerByPower.Trigger_Level));

            array_buffer[124] := TO_BYTE(SHR(TO_DWORD(buf1.TriggerByPower.PreTrigger_Amplitude), UINT#24));
            array_buffer[125] := TO_BYTE(SHR(TO_DWORD(buf1.TriggerByPower.PreTrigger_Amplitude), UINT#16));
            array_buffer[126] := TO_BYTE(SHR(TO_DWORD(buf1.TriggerByPower.PreTrigger_Amplitude),  UINT#8));
            array_buffer[127] := TO_BYTE(     TO_DWORD(buf1.TriggerByPower.PreTrigger_Amplitude));

            // ---- Misc: DINT ----
            array_buffer[128] := TO_BYTE(SHR(TO_DWORD(buf1.FreqCtrlMode), UINT#24));
            array_buffer[129] := TO_BYTE(SHR(TO_DWORD(buf1.FreqCtrlMode), UINT#16));
            array_buffer[130] := TO_BYTE(SHR(TO_DWORD(buf1.FreqCtrlMode),  UINT#8));
            array_buffer[131] := TO_BYTE(     TO_DWORD(buf1.FreqCtrlMode));

        END_METHOD

        METHOD PRIVATE buf2_TO_ByteArray
            VAR_IN_OUT
                buf2 : Axo_IQ_SeriesWelder_data2_136bytes;
                array_buffer : ARRAY[0..253] OF BYTE;
            END_VAR

            // ---- PowerReg (DINT → bytes 0..7) ----
            array_buffer[ 0] := TO_BYTE(SHR(TO_DWORD(buf2.PowerReg.PowerRegulationEnable), UINT#24));
            array_buffer[ 1] := TO_BYTE(SHR(TO_DWORD(buf2.PowerReg.PowerRegulationEnable), UINT#16));
            array_buffer[ 2] := TO_BYTE(SHR(TO_DWORD(buf2.PowerReg.PowerRegulationEnable),  UINT#8));
            array_buffer[ 3] := TO_BYTE(     TO_DWORD(buf2.PowerReg.PowerRegulationEnable));

            array_buffer[ 4] := TO_BYTE(SHR(TO_DWORD(buf2.PowerReg.PowerRegulationSetpoINT), UINT#24));
            array_buffer[ 5] := TO_BYTE(SHR(TO_DWORD(buf2.PowerReg.PowerRegulationSetpoINT), UINT#16));
            array_buffer[ 6] := TO_BYTE(SHR(TO_DWORD(buf2.PowerReg.PowerRegulationSetpoINT),  UINT#8));
            array_buffer[ 7] := TO_BYTE(     TO_DWORD(buf2.PowerReg.PowerRegulationSetpoINT));

            // ---- PressPretrigger.PreTriggerSource bits → bytes 8..11 ----
            array_buffer[ 8].%X0 := buf2.PressPretrigger.PreTriggerSource.bit24;
            array_buffer[ 8].%X1 := buf2.PressPretrigger.PreTriggerSource.bit25;
            array_buffer[ 8].%X2 := buf2.PressPretrigger.PreTriggerSource.bit26;
            array_buffer[ 8].%X3 := buf2.PressPretrigger.PreTriggerSource.bit27;
            array_buffer[ 8].%X4 := buf2.PressPretrigger.PreTriggerSource.bit28;
            array_buffer[ 8].%X5 := buf2.PressPretrigger.PreTriggerSource.bit29;
            array_buffer[ 8].%X6 := buf2.PressPretrigger.PreTriggerSource.bit30;
            array_buffer[ 8].%X7 := buf2.PressPretrigger.PreTriggerSource.bit31;

            array_buffer[ 9].%X0 := buf2.PressPretrigger.PreTriggerSource.bit16;
            array_buffer[ 9].%X1 := buf2.PressPretrigger.PreTriggerSource.bit17;
            array_buffer[ 9].%X2 := buf2.PressPretrigger.PreTriggerSource.bit18;
            array_buffer[ 9].%X3 := buf2.PressPretrigger.PreTriggerSource.bit19;
            array_buffer[ 9].%X4 := buf2.PressPretrigger.PreTriggerSource.bit20;
            array_buffer[ 9].%X5 := buf2.PressPretrigger.PreTriggerSource.bit21;
            array_buffer[ 9].%X6 := buf2.PressPretrigger.PreTriggerSource.bit22;
            array_buffer[ 9].%X7 := buf2.PressPretrigger.PreTriggerSource.bit23;

            array_buffer[10].%X0 := buf2.PressPretrigger.PreTriggerSource.bit8;
            array_buffer[10].%X1 := buf2.PressPretrigger.PreTriggerSource.bit9;
            array_buffer[10].%X2 := buf2.PressPretrigger.PreTriggerSource.bit10;
            array_buffer[10].%X3 := buf2.PressPretrigger.PreTriggerSource.bit11;
            array_buffer[10].%X4 := buf2.PressPretrigger.PreTriggerSource.bit12;
            array_buffer[10].%X5 := buf2.PressPretrigger.PreTriggerSource.bit13;
            array_buffer[10].%X6 := buf2.PressPretrigger.PreTriggerSource.bit14;
            array_buffer[10].%X7 := buf2.PressPretrigger.PreTriggerSource.bit15;

            array_buffer[11].%X0 := buf2.PressPretrigger.PreTriggerSource.AutoIn;
            array_buffer[11].%X1 := buf2.PressPretrigger.PreTriggerSource.Position_Switch;
            array_buffer[11].%X2 := buf2.PressPretrigger.PreTriggerSource._Time;
            array_buffer[11].%X3 := buf2.PressPretrigger.PreTriggerSource.Position;
            array_buffer[11].%X4 := buf2.PressPretrigger.PreTriggerSource.bit4;
            array_buffer[11].%X5 := buf2.PressPretrigger.PreTriggerSource.bit5;
            array_buffer[11].%X6 := buf2.PressPretrigger.PreTriggerSource.bit6;
            array_buffer[11].%X7 := buf2.PressPretrigger.PreTriggerSource.Enable_Trigger;

            // ---- PressPretrigger (DINTs → bytes 12..27) ----
            array_buffer[12] := TO_BYTE(SHR(TO_DWORD(buf2.PressPretrigger.Ignore1), UINT#24));
            array_buffer[13] := TO_BYTE(SHR(TO_DWORD(buf2.PressPretrigger.Ignore1), UINT#16));
            array_buffer[14] := TO_BYTE(SHR(TO_DWORD(buf2.PressPretrigger.Ignore1),  UINT#8));
            array_buffer[15] := TO_BYTE(     TO_DWORD(buf2.PressPretrigger.Ignore1));

            array_buffer[16] := TO_BYTE(SHR(TO_DWORD(buf2.PressPretrigger.Ignore2), UINT#24));
            array_buffer[17] := TO_BYTE(SHR(TO_DWORD(buf2.PressPretrigger.Ignore2), UINT#16));
            array_buffer[18] := TO_BYTE(SHR(TO_DWORD(buf2.PressPretrigger.Ignore2),  UINT#8));
            array_buffer[19] := TO_BYTE(     TO_DWORD(buf2.PressPretrigger.Ignore2));

            array_buffer[20] := TO_BYTE(SHR(TO_DWORD(buf2.PressPretrigger.PreTriggerTime), UINT#24));
            array_buffer[21] := TO_BYTE(SHR(TO_DWORD(buf2.PressPretrigger.PreTriggerTime), UINT#16));
            array_buffer[22] := TO_BYTE(SHR(TO_DWORD(buf2.PressPretrigger.PreTriggerTime),  UINT#8));
            array_buffer[23] := TO_BYTE(     TO_DWORD(buf2.PressPretrigger.PreTriggerTime));

            array_buffer[24] := TO_BYTE(SHR(TO_DWORD(buf2.PressPretrigger.PreTriggerPosition), UINT#24));
            array_buffer[25] := TO_BYTE(SHR(TO_DWORD(buf2.PressPretrigger.PreTriggerPosition), UINT#16));
            array_buffer[26] := TO_BYTE(SHR(TO_DWORD(buf2.PressPretrigger.PreTriggerPosition),  UINT#8));
            array_buffer[27] := TO_BYTE(     TO_DWORD(buf2.PressPretrigger.PreTriggerPosition));

            // ---- PressTrigger.TriggerSource bits → bytes 28..31 ----
            array_buffer[28].%X0 := buf2.PressTrigger.TriggerSource.res_bit24;
            array_buffer[28].%X1 := buf2.PressTrigger.TriggerSource.res_bit25;
            array_buffer[28].%X2 := buf2.PressTrigger.TriggerSource.res_bit26;
            array_buffer[28].%X3 := buf2.PressTrigger.TriggerSource.res_bit27;
            array_buffer[28].%X4 := buf2.PressTrigger.TriggerSource.res_bit28;
            array_buffer[28].%X5 := buf2.PressTrigger.TriggerSource.res_bit29;
            array_buffer[28].%X6 := buf2.PressTrigger.TriggerSource.res_bit30;
            array_buffer[28].%X7 := buf2.PressTrigger.TriggerSource.res_bit31;

            array_buffer[29].%X0 := buf2.PressTrigger.TriggerSource.res_bit16;
            array_buffer[29].%X1 := buf2.PressTrigger.TriggerSource.res_bit17;
            array_buffer[29].%X2 := buf2.PressTrigger.TriggerSource.res_bit18;
            array_buffer[29].%X3 := buf2.PressTrigger.TriggerSource.res_bit19;
            array_buffer[29].%X4 := buf2.PressTrigger.TriggerSource.res_bit20;
            array_buffer[29].%X5 := buf2.PressTrigger.TriggerSource.res_bit21;
            array_buffer[29].%X6 := buf2.PressTrigger.TriggerSource.res_bit22;
            array_buffer[29].%X7 := buf2.PressTrigger.TriggerSource.res_bit23;

            array_buffer[30].%X0 := buf2.PressTrigger.TriggerSource.res_bit8;
            array_buffer[30].%X1 := buf2.PressTrigger.TriggerSource.res_bit9;
            array_buffer[30].%X2 := buf2.PressTrigger.TriggerSource.res_bit10;
            array_buffer[30].%X3 := buf2.PressTrigger.TriggerSource.res_bit11;
            array_buffer[30].%X4 := buf2.PressTrigger.TriggerSource.res_bit12;
            array_buffer[30].%X5 := buf2.PressTrigger.TriggerSource.res_bit13;
            array_buffer[30].%X6 := buf2.PressTrigger.TriggerSource.res_bit14;
            array_buffer[30].%X7 := buf2.PressTrigger.TriggerSource.Enable_Trigger;

            array_buffer[31].%X0 := buf2.PressTrigger.TriggerSource.AutoIn;
            array_buffer[31].%X1 := buf2.PressTrigger.TriggerSource.Position_Switch;
            array_buffer[31].%X2 := buf2.PressTrigger.TriggerSource.res_bit2;
            array_buffer[31].%X3 := buf2.PressTrigger.TriggerSource.Position;
            array_buffer[31].%X4 := buf2.PressTrigger.TriggerSource.res_bit4;
            array_buffer[31].%X5 := buf2.PressTrigger.TriggerSource.Power;
            array_buffer[31].%X6 := buf2.PressTrigger.TriggerSource.res_bit6;
            array_buffer[31].%X7 := buf2.PressTrigger.TriggerSource.res_bit7;

            // ---- PressTrigger / Delay (DINTs → bytes 32..51) ----
            array_buffer[32] := TO_BYTE(SHR(TO_DWORD(buf2.PressTrigger.TriggerByPositionLevel), UINT#24));
            array_buffer[33] := TO_BYTE(SHR(TO_DWORD(buf2.PressTrigger.TriggerByPositionLevel), UINT#16));
            array_buffer[34] := TO_BYTE(SHR(TO_DWORD(buf2.PressTrigger.TriggerByPositionLevel),  UINT#8));
            array_buffer[35] := TO_BYTE(     TO_DWORD(buf2.PressTrigger.TriggerByPositionLevel));

            array_buffer[36] := TO_BYTE(SHR(TO_DWORD(buf2.PressTriggerDelay.TriggerDelaySource), UINT#24));
            array_buffer[37] := TO_BYTE(SHR(TO_DWORD(buf2.PressTriggerDelay.TriggerDelaySource), UINT#16));
            array_buffer[38] := TO_BYTE(SHR(TO_DWORD(buf2.PressTriggerDelay.TriggerDelaySource),  UINT#8));
            array_buffer[39] := TO_BYTE(     TO_DWORD(buf2.PressTriggerDelay.TriggerDelaySource));

            array_buffer[40] := TO_BYTE(SHR(TO_DWORD(buf2.PressTriggerDelay.TriggerDelayTimeout), UINT#24));
            array_buffer[41] := TO_BYTE(SHR(TO_DWORD(buf2.PressTriggerDelay.TriggerDelayTimeout), UINT#16));
            array_buffer[42] := TO_BYTE(SHR(TO_DWORD(buf2.PressTriggerDelay.TriggerDelayTimeout),  UINT#8));
            array_buffer[43] := TO_BYTE(     TO_DWORD(buf2.PressTriggerDelay.TriggerDelayTimeout));

            array_buffer[44] := TO_BYTE(SHR(TO_DWORD(buf2.PressTriggerDelay.TriggerDelayTime), UINT#24));
            array_buffer[45] := TO_BYTE(SHR(TO_DWORD(buf2.PressTriggerDelay.TriggerDelayTime), UINT#16));
            array_buffer[46] := TO_BYTE(SHR(TO_DWORD(buf2.PressTriggerDelay.TriggerDelayTime),  UINT#8));
            array_buffer[47] := TO_BYTE(     TO_DWORD(buf2.PressTriggerDelay.TriggerDelayTime));

            array_buffer[48] := TO_BYTE(SHR(TO_DWORD(buf2.PressTriggerDelay.TriggerDelayDistance), UINT#24));
            array_buffer[49] := TO_BYTE(SHR(TO_DWORD(buf2.PressTriggerDelay.TriggerDelayDistance), UINT#16));
            array_buffer[50] := TO_BYTE(SHR(TO_DWORD(buf2.PressTriggerDelay.TriggerDelayDistance),  UINT#8));
            array_buffer[51] := TO_BYTE(     TO_DWORD(buf2.PressTriggerDelay.TriggerDelayDistance));

            // ---- PressWeld.Weld1Source bits → bytes 52..55 ----
            array_buffer[52].%X0 := buf2.PressWeld.Weld1Source.bit24;
            array_buffer[52].%X1 := buf2.PressWeld.Weld1Source.bit25;
            array_buffer[52].%X2 := buf2.PressWeld.Weld1Source.bit26;
            array_buffer[52].%X3 := buf2.PressWeld.Weld1Source.bit27;
            array_buffer[52].%X4 := buf2.PressWeld.Weld1Source.bit28;
            array_buffer[52].%X5 := buf2.PressWeld.Weld1Source.bit29;
            array_buffer[52].%X6 := buf2.PressWeld.Weld1Source.bit30;
            array_buffer[52].%X7 := buf2.PressWeld.Weld1Source.bit31;

            array_buffer[53].%X0 := buf2.PressWeld.Weld1Source.bit16;
            array_buffer[53].%X1 := buf2.PressWeld.Weld1Source.bit17;
            array_buffer[53].%X2 := buf2.PressWeld.Weld1Source.bit18;
            array_buffer[53].%X3 := buf2.PressWeld.Weld1Source.bit19;
            array_buffer[53].%X4 := buf2.PressWeld.Weld1Source.bit20;
            array_buffer[53].%X5 := buf2.PressWeld.Weld1Source.bit21;
            array_buffer[53].%X6 := buf2.PressWeld.Weld1Source.bit22;
            array_buffer[53].%X7 := buf2.PressWeld.Weld1Source.bit23;

            array_buffer[54].%X0 := buf2.PressWeld.Weld1Source.bit8;
            array_buffer[54].%X1 := buf2.PressWeld.Weld1Source.bit9;
            array_buffer[54].%X2 := buf2.PressWeld.Weld1Source.bit10;
            array_buffer[54].%X3 := buf2.PressWeld.Weld1Source.bit11;
            array_buffer[54].%X4 := buf2.PressWeld.Weld1Source.bit12;
            array_buffer[54].%X5 := buf2.PressWeld.Weld1Source.bit13;
            array_buffer[54].%X6 := buf2.PressWeld.Weld1Source.bit14;
            array_buffer[54].%X7 := buf2.PressWeld.Weld1Source.Enable_Weld_1;

            array_buffer[55].%X0 := buf2.PressWeld.Weld1Source._Time;
            array_buffer[55].%X1 := buf2.PressWeld.Weld1Source.Power;
            array_buffer[55].%X2 := buf2.PressWeld.Weld1Source.Energy;
            array_buffer[55].%X3 := buf2.PressWeld.Weld1Source.Distance;
            array_buffer[55].%X4 := buf2.PressWeld.Weld1Source.Position;
            array_buffer[55].%X5 := buf2.PressWeld.Weld1Source.Ground_Detect;
            array_buffer[55].%X6 := buf2.PressWeld.Weld1Source.Force;
            array_buffer[55].%X7 := buf2.PressWeld.Weld1Source.bit7;

            // ---- PressWeld (DINTs → bytes 56..67) ----
            array_buffer[56] := TO_BYTE(SHR(TO_DWORD(buf2.PressWeld.Weld1Timeout), UINT#24));
            array_buffer[57] := TO_BYTE(SHR(TO_DWORD(buf2.PressWeld.Weld1Timeout), UINT#16));
            array_buffer[58] := TO_BYTE(SHR(TO_DWORD(buf2.PressWeld.Weld1Timeout),  UINT#8));
            array_buffer[59] := TO_BYTE(     TO_DWORD(buf2.PressWeld.Weld1Timeout));

            array_buffer[60] := TO_BYTE(SHR(TO_DWORD(buf2.PressWeld.Weld1Distance), UINT#24));
            array_buffer[61] := TO_BYTE(SHR(TO_DWORD(buf2.PressWeld.Weld1Distance), UINT#16));
            array_buffer[62] := TO_BYTE(SHR(TO_DWORD(buf2.PressWeld.Weld1Distance),  UINT#8));
            array_buffer[63] := TO_BYTE(     TO_DWORD(buf2.PressWeld.Weld1Distance));

            array_buffer[64] := TO_BYTE(SHR(TO_DWORD(buf2.PressWeld.Weld1Position), UINT#24));
            array_buffer[65] := TO_BYTE(SHR(TO_DWORD(buf2.PressWeld.Weld1Position), UINT#16));
            array_buffer[66] := TO_BYTE(SHR(TO_DWORD(buf2.PressWeld.Weld1Position),  UINT#8));
            array_buffer[67] := TO_BYTE(     TO_DWORD(buf2.PressWeld.Weld1Position));

            // ---- PressWeld.Weld2Source bits → bytes 68..71 ----
            array_buffer[68].%X0 := buf2.PressWeld.Weld2Source.bit24;
            array_buffer[68].%X1 := buf2.PressWeld.Weld2Source.bit25;
            array_buffer[68].%X2 := buf2.PressWeld.Weld2Source.bit26;
            array_buffer[68].%X3 := buf2.PressWeld.Weld2Source.bit27;
            array_buffer[68].%X4 := buf2.PressWeld.Weld2Source.bit28;
            array_buffer[68].%X5 := buf2.PressWeld.Weld2Source.bit29;
            array_buffer[68].%X6 := buf2.PressWeld.Weld2Source.bit30;
            array_buffer[68].%X7 := buf2.PressWeld.Weld2Source.bit31;

            array_buffer[69].%X0 := buf2.PressWeld.Weld2Source.bit16;
            array_buffer[69].%X1 := buf2.PressWeld.Weld2Source.bit17;
            array_buffer[69].%X2 := buf2.PressWeld.Weld2Source.bit18;
            array_buffer[69].%X3 := buf2.PressWeld.Weld2Source.bit19;
            array_buffer[69].%X4 := buf2.PressWeld.Weld2Source.bit20;
            array_buffer[69].%X5 := buf2.PressWeld.Weld2Source.bit21;
            array_buffer[69].%X6 := buf2.PressWeld.Weld2Source.bit22;
            array_buffer[69].%X7 := buf2.PressWeld.Weld2Source.bit23;

            array_buffer[70].%X0 := buf2.PressWeld.Weld2Source.bit8;
            array_buffer[70].%X1 := buf2.PressWeld.Weld2Source.bit9;
            array_buffer[70].%X2 := buf2.PressWeld.Weld2Source.bit10;
            array_buffer[70].%X3 := buf2.PressWeld.Weld2Source.bit11;
            array_buffer[70].%X4 := buf2.PressWeld.Weld2Source.bit12;
            array_buffer[70].%X5 := buf2.PressWeld.Weld2Source.bit13;
            array_buffer[70].%X6 := buf2.PressWeld.Weld2Source.bit14;
            array_buffer[70].%X7 := buf2.PressWeld.Weld2Source.Enable_Weld_1;

            array_buffer[71].%X0 := buf2.PressWeld.Weld2Source._Time;
            array_buffer[71].%X1 := buf2.PressWeld.Weld2Source.Power;
            array_buffer[71].%X2 := buf2.PressWeld.Weld2Source.Energy;
            array_buffer[71].%X3 := buf2.PressWeld.Weld2Source.Distance;
            array_buffer[71].%X4 := buf2.PressWeld.Weld2Source.Position;
            array_buffer[71].%X5 := buf2.PressWeld.Weld2Source.Ground_Detect;
            array_buffer[71].%X6 := buf2.PressWeld.Weld2Source.Force;
            array_buffer[71].%X7 := buf2.PressWeld.Weld2Source.bit7;

            // ---- PressWeld (DINTs → bytes 72..99) ----
            array_buffer[72] := TO_BYTE(SHR(TO_DWORD(buf2.PressWeld.Weld2SecondarySource), UINT#24));
            array_buffer[73] := TO_BYTE(SHR(TO_DWORD(buf2.PressWeld.Weld2SecondarySource), UINT#16));
            array_buffer[74] := TO_BYTE(SHR(TO_DWORD(buf2.PressWeld.Weld2SecondarySource),  UINT#8));
            array_buffer[75] := TO_BYTE(     TO_DWORD(buf2.PressWeld.Weld2SecondarySource));

            array_buffer[76] := TO_BYTE(SHR(TO_DWORD(buf2.PressWeld.Weld2Timeout), UINT#24));
            array_buffer[77] := TO_BYTE(SHR(TO_DWORD(buf2.PressWeld.Weld2Timeout), UINT#16));
            array_buffer[78] := TO_BYTE(SHR(TO_DWORD(buf2.PressWeld.Weld2Timeout),  UINT#8));
            array_buffer[79] := TO_BYTE(     TO_DWORD(buf2.PressWeld.Weld2Timeout));

            array_buffer[80] := TO_BYTE(SHR(TO_DWORD(buf2.PressWeld.Weld2Time), UINT#24));
            array_buffer[81] := TO_BYTE(SHR(TO_DWORD(buf2.PressWeld.Weld2Time), UINT#16));
            array_buffer[82] := TO_BYTE(SHR(TO_DWORD(buf2.PressWeld.Weld2Time),  UINT#8));
            array_buffer[83] := TO_BYTE(     TO_DWORD(buf2.PressWeld.Weld2Time));

            array_buffer[84] := TO_BYTE(SHR(TO_DWORD(buf2.PressWeld.Weld2Energy), UINT#24));
            array_buffer[85] := TO_BYTE(SHR(TO_DWORD(buf2.PressWeld.Weld2Energy), UINT#16));
            array_buffer[86] := TO_BYTE(SHR(TO_DWORD(buf2.PressWeld.Weld2Energy),  UINT#8));
            array_buffer[87] := TO_BYTE(     TO_DWORD(buf2.PressWeld.Weld2Energy));

            array_buffer[88] := TO_BYTE(SHR(TO_DWORD(buf2.PressWeld.Weld2Power), UINT#24));
            array_buffer[89] := TO_BYTE(SHR(TO_DWORD(buf2.PressWeld.Weld2Power), UINT#16));
            array_buffer[90] := TO_BYTE(SHR(TO_DWORD(buf2.PressWeld.Weld2Power),  UINT#8));
            array_buffer[91] := TO_BYTE(     TO_DWORD(buf2.PressWeld.Weld2Power));

            array_buffer[92] := TO_BYTE(SHR(TO_DWORD(buf2.PressWeld.Weld2Distance), UINT#24));
            array_buffer[93] := TO_BYTE(SHR(TO_DWORD(buf2.PressWeld.Weld2Distance), UINT#16));
            array_buffer[94] := TO_BYTE(SHR(TO_DWORD(buf2.PressWeld.Weld2Distance),  UINT#8));
            array_buffer[95] := TO_BYTE(     TO_DWORD(buf2.PressWeld.Weld2Distance));

            array_buffer[96] := TO_BYTE(SHR(TO_DWORD(buf2.PressWeld.Weld2Position), UINT#24));
            array_buffer[97] := TO_BYTE(SHR(TO_DWORD(buf2.PressWeld.Weld2Position), UINT#16));
            array_buffer[98] := TO_BYTE(SHR(TO_DWORD(buf2.PressWeld.Weld2Position),  UINT#8));
            array_buffer[99] := TO_BYTE(     TO_DWORD(buf2.PressWeld.Weld2Position));

            // ---- PressWeldScrub (DINTs → bytes 100..107) ----
            array_buffer[100] := TO_BYTE(SHR(TO_DWORD(buf2.PressWeldScrub.ScrubMode), UINT#24));
            array_buffer[101] := TO_BYTE(SHR(TO_DWORD(buf2.PressWeldScrub.ScrubMode), UINT#16));
            array_buffer[102] := TO_BYTE(SHR(TO_DWORD(buf2.PressWeldScrub.ScrubMode),  UINT#8));
            array_buffer[103] := TO_BYTE(     TO_DWORD(buf2.PressWeldScrub.ScrubMode));

            array_buffer[104] := TO_BYTE(SHR(TO_DWORD(buf2.PressWeldScrub.ScrubTime), UINT#24));
            array_buffer[105] := TO_BYTE(SHR(TO_DWORD(buf2.PressWeldScrub.ScrubTime), UINT#16));
            array_buffer[106] := TO_BYTE(SHR(TO_DWORD(buf2.PressWeldScrub.ScrubTime),  UINT#8));
            array_buffer[107] := TO_BYTE(     TO_DWORD(buf2.PressWeldScrub.ScrubTime));

            // ---- PressPostWeld.DynamicHoldMode bits → bytes 108..111 ----
            array_buffer[108].%X0 := buf2.PressPostWeld.DynamicHoldMode.bit24;
            array_buffer[108].%X1 := buf2.PressPostWeld.DynamicHoldMode.bit25;
            array_buffer[108].%X2 := buf2.PressPostWeld.DynamicHoldMode.bit26;
            array_buffer[108].%X3 := buf2.PressPostWeld.DynamicHoldMode.bit27;
            array_buffer[108].%X4 := buf2.PressPostWeld.DynamicHoldMode.bit28;
            array_buffer[108].%X5 := buf2.PressPostWeld.DynamicHoldMode.bit29;
            array_buffer[108].%X6 := buf2.PressPostWeld.DynamicHoldMode.bit30;
            array_buffer[108].%X7 := buf2.PressPostWeld.DynamicHoldMode.bit31;

            array_buffer[109].%X0 := buf2.PressPostWeld.DynamicHoldMode.bit16;
            array_buffer[109].%X1 := buf2.PressPostWeld.DynamicHoldMode.bit17;
            array_buffer[109].%X2 := buf2.PressPostWeld.DynamicHoldMode.bit18;
            array_buffer[109].%X3 := buf2.PressPostWeld.DynamicHoldMode.bit19;
            array_buffer[109].%X4 := buf2.PressPostWeld.DynamicHoldMode.bit20;
            array_buffer[109].%X5 := buf2.PressPostWeld.DynamicHoldMode.bit21;
            array_buffer[109].%X6 := buf2.PressPostWeld.DynamicHoldMode.bit22;
            array_buffer[109].%X7 := buf2.PressPostWeld.DynamicHoldMode.bit23;

            array_buffer[110].%X0 := buf2.PressPostWeld.DynamicHoldMode.bit8;
            array_buffer[110].%X1 := buf2.PressPostWeld.DynamicHoldMode.bit9;
            array_buffer[110].%X2 := buf2.PressPostWeld.DynamicHoldMode.bit10;
            array_buffer[110].%X3 := buf2.PressPostWeld.DynamicHoldMode.bit11;
            array_buffer[110].%X4 := buf2.PressPostWeld.DynamicHoldMode.bit12;
            array_buffer[110].%X5 := buf2.PressPostWeld.DynamicHoldMode.bit13;
            array_buffer[110].%X6 := buf2.PressPostWeld.DynamicHoldMode.bit14;
            array_buffer[110].%X7 := buf2.PressPostWeld.DynamicHoldMode.bit15;

            array_buffer[111].%X0 := buf2.PressPostWeld.DynamicHoldMode._Time;
            array_buffer[111].%X1 := buf2.PressPostWeld.DynamicHoldMode.Distance;
            array_buffer[111].%X2 := buf2.PressPostWeld.DynamicHoldMode.Force;
            array_buffer[111].%X3 := buf2.PressPostWeld.DynamicHoldMode.AutoIn;
            array_buffer[111].%X4 := buf2.PressPostWeld.DynamicHoldMode.Velocity;
            array_buffer[111].%X5 := buf2.PressPostWeld.DynamicHoldMode.bit5;
            array_buffer[111].%X6 := buf2.PressPostWeld.DynamicHoldMode.bit6;
            array_buffer[111].%X7 := buf2.PressPostWeld.DynamicHoldMode.bit7;

            // ---- PressPostWeld (DINTs → bytes 112..135) ----
            array_buffer[112] := TO_BYTE(SHR(TO_DWORD(buf2.PressPostWeld.DynamicHoldTimeout), UINT#24));
            array_buffer[113] := TO_BYTE(SHR(TO_DWORD(buf2.PressPostWeld.DynamicHoldTimeout), UINT#16));
            array_buffer[114] := TO_BYTE(SHR(TO_DWORD(buf2.PressPostWeld.DynamicHoldTimeout),  UINT#8));
            array_buffer[115] := TO_BYTE(     TO_DWORD(buf2.PressPostWeld.DynamicHoldTimeout));

            array_buffer[116] := TO_BYTE(SHR(TO_DWORD(buf2.PressPostWeld.DynamicHoldDistance), UINT#24));
            array_buffer[117] := TO_BYTE(SHR(TO_DWORD(buf2.PressPostWeld.DynamicHoldDistance), UINT#16));
            array_buffer[118] := TO_BYTE(SHR(TO_DWORD(buf2.PressPostWeld.DynamicHoldDistance),  UINT#8));
            array_buffer[119] := TO_BYTE(     TO_DWORD(buf2.PressPostWeld.DynamicHoldDistance));

            array_buffer[120] := TO_BYTE(SHR(TO_DWORD(buf2.PressPostWeld.DynamicHoldForce), UINT#24));
            array_buffer[121] := TO_BYTE(SHR(TO_DWORD(buf2.PressPostWeld.DynamicHoldForce), UINT#16));
            array_buffer[122] := TO_BYTE(SHR(TO_DWORD(buf2.PressPostWeld.DynamicHoldForce),  UINT#8));
            array_buffer[123] := TO_BYTE(     TO_DWORD(buf2.PressPostWeld.DynamicHoldForce));

            array_buffer[124] := TO_BYTE(SHR(TO_DWORD(buf2.PressPostWeld.StaticHoldMode), UINT#24));
            array_buffer[125] := TO_BYTE(SHR(TO_DWORD(buf2.PressPostWeld.StaticHoldMode), UINT#16));
            array_buffer[126] := TO_BYTE(SHR(TO_DWORD(buf2.PressPostWeld.StaticHoldMode),  UINT#8));
            array_buffer[127] := TO_BYTE(     TO_DWORD(buf2.PressPostWeld.StaticHoldMode));
